// TIA Portal V20 program export: 31 tag tables, 33 data types, 19 data blocks, 74 code blocks (in call order from the OBs), 22 instance data blocks

VAR_GLOBAL   // PLC tag table "Default tag table"
   System_Byte AT %MB1 : Byte;
   FirstScan AT %M1.0 : Bool;
   DiagStatusUpdate AT %M1.1 : Bool;
   AlwaysTRUE AT %M1.2 : Bool;
   AlwaysFALSE AT %M1.3 : Bool;
   Clock_Byte AT %MB0 : Byte;
   Clock_10Hz AT %M0.0 : Bool;
   Clock_5Hz AT %M0.1 : Bool;
   "Clock_2.5Hz" AT %M0.2 : Bool;
   Clock_2Hz AT %M0.3 : Bool;
   "Clock_1.25Hz" AT %M0.4 : Bool;
   Clock_1Hz AT %M0.5 : Bool;
   "Clock_0.625Hz" AT %M0.6 : Bool;
   "Clock_0.5Hz" AT %M0.7 : Bool;
   startBit AT %M100.0 : Bool;
   stopBit AT %M100.1 : Bool;
   ResetBit AT %M100.2 : Bool;
END_VAR

VAR_GLOBAL   // PLC tag table "Tag table_1"
END_VAR

VAR_GLOBAL   // PLC tag table "Default tag table_1"
END_VAR

VAR_GLOBAL   // PLC tag table "ConvConstantEmptyLine"
END_VAR
VAR_GLOBAL CONSTANT   // user constants
   minEmptyLine : Int := 2001;
   maxEmptyLine : Int := 2109;
   "J1.1.1" : Int := 2001;   // J1.1.1
   "J1.1.2" : Int := 2002;   // J1.1.2
   "J1.1.3" : Int := 2003;   // J1.1.3
   "J1.1.4" : Int := 2004;   // J1.1.4
   "J1.1.5" : Int := 2005;   // J1.1.5
   "J1.1.6" : Int := 2006;   // J1.1.6
   "J1.1.7" : Int := 2007;   // J1.1.7
   "J1.1.8" : Int := 2008;   // J1.1.8
   "J1.1.9" : Int := 2009;   // J1.1.9
   "J1.1.10" : Int := 2010;   // J1.1.10
   "J1.1.11" : Int := 2011;   // J1.1.11
   "J1.1.12" : Int := 2012;   // J1.1.12
   "J1.1.13" : Int := 2013;   // J1.1.13
   "J1.1.14" : Int := 2014;   // J1.1.14
   "J1.1.15" : Int := 2015;   // J1.1.15
   "J1.2.1" : Int := 2016;   // J1.2.1
   "J1.2.2" : Int := 2017;   // J1.2.2
   "J1.2.3" : Int := 2018;   // J1.2.3 Staright for Merger1
   "J2.1.1" : Int := 2019;   // J2.1.1
   "J2.1.2" : Int := 2020;   // J2.1.2
   "J2.1.3" : Int := 2021;   // J2.1.3
   "J2.1.4" : Int := 2022;   // J2.1.4
   "J2.1.5" : Int := 2023;   // J2.1.5
   "J2.1.6" : Int := 2024;   // J2.1.6
   "J2.1.7" : Int := 2025;   // J2.1.7
   "J2.1.8" : Int := 2026;   // J2.1.8
   "J2.1.9" : Int := 2027;   // J2.1.9
   "J2.1.10" : Int := 2028;   // J2.1.10
   "J2.1.11" : Int := 2029;   // J2.1.11
   "J2.1.12" : Int := 2030;   // J2.1.12
   "J2.1.13" : Int := 2031;   // J2.1.13
   "J2.1.14" : Int := 2032;   // J2.1.14
   "J2.1.15" : Int := 2033;   // J2.1.15
   "J2.2.1" : Int := 2034;   // J2.2.1
   "J2.2.2" : Int := 2035;   // J2.2.2
   "J2.3.1" : Int := 2036;   // J2.3.1
   "J2.4.1" : Int := 2037;   // J2.4.1 Arm for Merger1
   "J1.2.4" : Int := 2038;   // J1.2.4 Merger 1
   "J1.2.5" : Int := 2039;   // J1.2.5
   "J1.3.1" : Int := 2040;   // J1.3.1
   "J1.3.2" : Int := 2041;   // J1.3.2
   "J1.4.1" : Int := 2042;   // J1.4.1
   "J1.4.2" : Int := 2043;   // J1.4.2
   "J1.4.3" : Int := 2044;   // J1.4.3
   "J1.4.4" : Int := 2045;   // J1.4.4
   "J1.4.5" : Int := 2046;   // J1.4.5
   "J1.4.6" : Int := 2047;   // J1.4.6
   "J1.4.7" : Int := 2048;   // J1.4.7
   "J1.5.1" : Int := 2049;   // J1.5.1
   "J1.5.2" : Int := 2050;   // J1.5.2
   "J1.5.3" : Int := 2051;   // J1.5.3
   "J1.5.4" : Int := 2052;   // J1.5.4
   "J1.7.1" : Int := 2053;   // J1.7.1 (Go straight )
   "J1.7.2" : Int := 2054;   // J1.7.2
   "J1.8.1" : Int := 2055;   // J1.8.1
   "J1.8.2" : Int := 2056;   // J1.8.2
   "J1.9.1" : Int := 2057;   // J1.9.1
   "J1.10.1" : Int := 2058;   // J1.10.1
   "J1.11.1" : Int := 2059;   // J1.11.1
   "J1.11.2" : Int := 2060;   // J1.11.2
   "J1.11.3" : Int := 2061;   // J1.11.3
   "J1.11.4" : Int := 2062;   // J1.11.4
   "J1.11.5" : Int := 2063;   // J1.11.5
   "J1.11.6" : Int := 2064;   // J1.11.6
   "J1.11.7" : Int := 2065;   // J1.11.7
   "J1.11.8" : Int := 2066;   // J1.11.8
   "J1.11.9" : Int := 2067;   // J1.11.9
   "J1.11.10" : Int := 2068;   // J1.11.10
   "J1.11.11" : Int := 2069;   // J1.11.11
   "J1.11.12" : Int := 2070;   // J1.11.12
   "J1.11.13" : Int := 2071;   // J1.11.13
   "K1.1.1" : Int := 2072;   // K1.1.1 (Go Left)
   "K1.2.1" : Int := 2073;   // K1.2.1
   "K1.3.1" : Int := 2074;   // K1.3.1
   "K1.4.1" : Int := 2075;   // K1.4.1
   "K1.4.2" : Int := 2076;   // K1.4.2
   "K1.4.3" : Int := 2077;   // K1.4.3
   "K1.4.4" : Int := 2078;   // K1.4.4
   "K1.4.5" : Int := 2079;   // K1.4.5
   "K1.4.6" : Int := 2080;   // K1.4.6
   "K1.4.7" : Int := 2081;   // K1.4.7
   "K1.4.8" : Int := 2082;   // K1.4.8
   "K1.4.9" : Int := 2083;   // K1.4.9
   "K1.4.10" : Int := 2084;   // K1.4.10
   "K1.5.1" : Int := 2085;   // K1.5.1
   "K1.5.2" : Int := 2086;   // K1.5.2
   "K1.5.3" : Int := 2087;   // K1.5.3
   "K1.5.4" : Int := 2088;   // K1.5.4
   "K1.5.5" : Int := 2089;   // K1.5.5
   "K1.5.6" : Int := 2090;   // K1.5.6
   "K1.5.7" : Int := 2091;   // K1.5.7
   "K1.5.8" : Int := 2092;   // K1.5.8
   "K1.6.1" : Int := 2093;   // K1.6.1
   "K1.6.2" : Int := 2094;   // K1.6.2
   "K1.7.1" : Int := 2095;   // K1.7.1
   "K1.7.2" : Int := 2096;   // K1.7.2
   "K1.8.1" : Int := 2097;   // K1.8.1
   "K1.8.2" : Int := 2098;   // K1.8.2
   "K1.8.3" : Int := 2099;   // K1.8.3
   "K1.9.1" : Int := 2100;   // K1.9.1
   "K1.9.2" : Int := 2101;   // K1.9.2
   "K1.9.3" : Int := 2102;   // K1.9.3
   "K1.9.4" : Int := 2103;   // K1.9.4
   "K1.9.5" : Int := 2104;   // K1.9.5
   "K1.9.6" : Int := 2105;   // K1.9.6
   "K1.9.7" : Int := 2106;   // K1.9.7
   "K1.10.1" : Int := 2107;   // K1.10.1
   "J1.6.1" : Int := 2108;   // Mabs J1.6.1
   "J1.6.2" : Int := 2109;   // Mabs J1.6.2
END_VAR

VAR_GLOBAL   // PLC tag table "MabsEmptyLine"
   "MABS_J1.6.1_IN" AT %I839.0 : "Global.IB_P01_02_03_in_64bytes_struct";
   "MABS_J1.6.1_Out" AT %Q761.0 : "Global.IB_P01_02_03_out_64bytes_struct";
   "MABS_J1.6.2_IN" AT %I903.0 : "Global.IB_P01_02_03_in_64bytes_struct";
   "MABS_J1.6.2_Out" AT %Q825.0 : "Global.IB_P01_02_03_out_64bytes_struct";
END_VAR

VAR_GLOBAL   // PLC tag table "ASi Alarm"
   "BW_ASi23 -MCC100 -210KE3 -ConfigErr_Circuit1_Slave(16-31)A" AT %IW2366 : Word;
   "BW_ASi23 -MCC100 -210KE3 -ConfigErr_Circuit1_Slave(16-31)B" AT %IW2370 : Word;
   "BW_ASi23 -MCC100 -210KE3 -PeriErr_Circuit1_Slave(16-31)A" AT %IW2374 : Word;
   "BW_ASi23 -MCC100 -210KE3 -PeriErr_Circuit1_Slave(16-31)B" AT %IW2378 : Word;
   "BW_ASi23 -MCC100 -210KE3 -ConfigErr_Circuit2_Slave(0-15)A" AT %IW2380 : Word;
   "BW_ASi23 -MCC100 -210KE3 -ConfigErr_Circuit2_Slave(16-31)A" AT %IW2382 : Word;
   "BW_ASi23 -MCC100 -210KE3 -ConfigErr_Circuit2_Slave(0-15)B" AT %IW2384 : Word;
   "BW_ASi23 -MCC100 -210KE3 -ConfigErr_Circuit2_Slave(16-31)B" AT %IW2386 : Word;
   "BW_ASi23 -MCC100 -210KE3 -PeriErr_Circuit2_Slave(0-15)A" AT %IW2388 : Word;
   "BW_ASi23 -MCC100 -210KE3 -PeriErr_Circuit2_Slave(16-31)A" AT %IW2390 : Word;
   "BW_ASi23 -MCC100 -210KE3 -PeriErr_Circuit2_Slave(0-15)B" AT %IW2392 : Word;
   "BW_ASi23 -MCC100 -210KE3 -PeriErr_Circuit2_Slave(16-31)B" AT %IW2394 : Word;
   "BW_ASi23 -MCC100 -210KE3 -ConfigErr_Circuit1_Slave(0-15)A" AT %IW2364 : Word;
   "BW_ASi23 -MCC100 -210KE3 -ConfigErr_Circuit1_Slave(0-15)B" AT %IW2368 : Word;
   "BW_ASi23 -MCC100 -210KE3 -PeriErr_Circuit1_Slave(0-15)A" AT %IW2372 : Word;
   "BW_ASi23 -MCC100 -210KE3 -PeriErr_Circuit1_Slave(0-15)B" AT %IW2376 : Word;
END_VAR

VAR_GLOBAL   // PLC tag table "ASi"
   "ASiGW-MCC100-bw23-C1: Input" AT %I2300.0 : "tASiGW-MCC100-bw23-C1: Input";
   "ASiGW-MCC100-bw23-C1: Output" AT %Q2300.0 : "tASiGW-MCC100-bw23-C1: Output";
   "ASiGW-MCC100-bw23-C1: ConfigErr" AT %I2364.0 : "Config/PeriErr";
   "ASiGW-MCC100-bw23-C1: PeriErr" AT %I2372.0 : "Config/PeriErr";
END_VAR

VAR_GLOBAL   // PLC tag table "Circuit Breaker"
END_VAR

VAR_GLOBAL   // PLC tag table "ConvConstant"
END_VAR
VAR_GLOBAL CONSTANT   // user constants
   gMinA1 : Int := 1001;
   gMaxA1 : Int := 1002;
   gMinB1 : Int := 2001;
   gMaxB1 : Int := 2002;
   gMinC1 : Int := 3001;
   gMaxC1 : Int := 3054;
   gMinD1 : Int := 4001;
   gMaxD1 : Int := 4002;
END_VAR

VAR_GLOBAL   // PLC tag table "DM262"
   "Dataman-TriggerEnable" AT %Q10.0 : Bool;
   "Dataman-Trigger" AT %Q10.1 : Bool;
   "Dataman-TriggerReady" AT %I10.0 : Bool;
   "Dataman-TriggerAck" AT %I10.1 : Bool;
   "Dataman-Acquiring" AT %I10.2 : Bool;
   "Dataman-MissedAcq" AT %I10.3 : Bool;
   "Dataman-TriggerID" AT %IW11 : Word;
   "Dataman-BufferResultsEnable" AT %Q11.0 : Bool;
   "Dataman-ResultsAck" AT %Q11.1 : Bool;
   "Dataman-Decoding" AT %I13.0 : Bool;
   "Dataman-Decode Complete" AT %I13.1 : Bool;
   "Dataman-Results Buffer Overrun" AT %I13.2 : Bool;
   "Dataman-Results Available" AT %I13.3 : Bool;
   "Dataman-General Fault" AT %I13.7 : Bool;
   "Dataman-Train Code" AT %Q12.0 : Bool;
   "Dataman-Train Match String" AT %Q12.1 : Bool;
   "Dataman-Train Focus" AT %Q12.2 : Bool;
   "Dataman-Train Brightness" AT %Q12.3 : Bool;
   "Dataman-Untrain" AT %Q12.4 : Bool;
   "Dataman-Execute DMCC" AT %Q12.6 : Bool;
   "Dataman-Set Match String" AT %Q12.7 : Bool;
   "Dataman-Train Code Ack" AT %I14.0 : Bool;
   "Dataman-Train Match String Ack" AT %I14.1 : Bool;
   "Dataman-Train Focus Ack" AT %I14.2 : Bool;
   "Dataman-Train Brightness Ack" AT %I14.3 : Bool;
   "Dataman-Untrain Ack" AT %I14.4 : Bool;
   "Dataman-Execute DMCC Ack" AT %I14.6 : Bool;
   "Dataman-Set Match String Ack" AT %I14.7 : Bool;
   "Dataman-UserData Option" AT %QW13 : Word;
   "Dataman-UserData Length" AT %QW15 : Word;
   "Dataman-UserData[0]" AT %QB17 : Byte;
   "Dataman-UserData[1]" AT %QB18 : Byte;
   "Dataman-UserData[2]" AT %QB19 : Byte;
   "Dataman-UserData[3]" AT %QB20 : Byte;
   "Dataman-UserData[4]" AT %QB21 : Byte;
   "Dataman-UserData[5]" AT %QB22 : Byte;
   "Dataman-UserData[6]" AT %QB23 : Byte;
   "Dataman-UserData[7]" AT %QB24 : Byte;
   "Dataman-UserData[8]" AT %QB25 : Byte;
   "Dataman-UserData[9]" AT %QB26 : Byte;
   "Dataman-UserData[10]" AT %QB27 : Byte;
   "Dataman-UserData[11]" AT %QB28 : Byte;
   "Dataman-UserData[12]" AT %QB29 : Byte;
   "Dataman-UserData[13]" AT %QB30 : Byte;
   "Dataman-UserData[14]" AT %QB31 : Byte;
   "Dataman-UserData[15]" AT %QB32 : Byte;
   "Dataman-ResultID" AT %IW15 : Word;
   "Dataman-Result Code" AT %IW18 : Word;
   "Dataman-Read / No Read" AT %I18.0 : Bool;
   "Dataman-Validated / Not Validated" AT %I18.1 : Bool;
   "Dataman-Verified / Not Verified" AT %I18.2 : Bool;
   "Dataman-Acquisition Trigger Overrun" AT %I18.3 : Bool;
   "Dataman-Acquisition Buffer Overflow" AT %I18.4 : Bool;
   "Dataman-Result Extended" AT %IW19 : Word;
   "Dataman-Result Length" AT %IW21 : Word;
   "Dataman-InspectionResults[0]" AT %IB23 : Byte;
   "Dataman-InspectionResults[1]" AT %IB24 : Byte;
   "Dataman-InspectionResults[2]" AT %IB25 : Byte;
   "Dataman-InspectionResults[3]" AT %IB26 : Byte;
   "Dataman-InspectionResults[4]" AT %IB27 : Byte;
   "Dataman-InspectionResults[5]" AT %IB28 : Byte;
   "Dataman-InspectionResults[6]" AT %IB29 : Byte;
   "Dataman-InspectionResults[7]" AT %IB30 : Byte;
   "Dataman-InspectionResults[8]" AT %IB31 : Byte;
   "Dataman-InspectionResults[9]" AT %IB32 : Byte;
   "Dataman-InspectionResults[10]" AT %IB33 : Byte;
   "Dataman-InspectionResults[11]" AT %IB34 : Byte;
   "Dataman-InspectionResults[12]" AT %IB35 : Byte;
   "Dataman-InspectionResults[13]" AT %IB36 : Byte;
   "Dataman-InspectionResults[14]" AT %IB37 : Byte;
   "Dataman-InspectionResults[15]" AT %IB38 : Byte;
   "Result Data" AT %I23.0 : "Global.BarCode";
   "User Data" AT %Q17.0 : "Global.BarCode";
END_VAR

VAR_GLOBAL   // PLC tag table "Default tag table_3"
END_VAR

VAR_GLOBAL   // PLC tag table "Klaxon"
END_VAR

VAR_GLOBAL   // PLC tag table "SSR"
END_VAR

VAR_GLOBAL   // PLC tag table "Safety"
END_VAR

VAR_GLOBAL   // PLC tag table "ConvConstantA1"
END_VAR
VAR_GLOBAL CONSTANT   // user constants
   minA1 : Int := 1001;
   maxA1 : Int := 1002;
END_VAR

VAR_GLOBAL   // PLC tag table "ConvConstantB1"
END_VAR
VAR_GLOBAL CONSTANT   // user constants
   minB1 : Int := 2001;
   maxB1 : Int := 2002;
END_VAR

VAR_GLOBAL   // PLC tag table "Default tag table_2"
END_VAR

VAR_GLOBAL   // PLC tag table "ConvConstantC1"
END_VAR
VAR_GLOBAL CONSTANT   // user constants
   minC1 : Int := 3001;
   maxC1 : Int := 3054;
   "Conveyor_C1.1.1" : Int := 3001;
   "Conveyor_C1.1.2" : Int := 3002;
   "Conveyor_C1.1.3" : Int := 3003;
   "MABS_C1.2.1" : Int := 3051;
   "MABS_C1.2.2" : Int := 3052;
   "Conveyor_C1.9.1" : Int := 3031;
   "Conveyor_C1.10.1" : Int := 3032;
   "Conveyor_C1.11.1" : Int := 3033;
   "Conveyor_C1.11.2" : Int := 3034;
   "Conveyor_C1.12.1" : Int := 3035;
   "Conveyor_C1.12.2" : Int := 3036;
   "Conveyor_C1.12.3" : Int := 3037;
   "Transfer_C1.13.1" : Int := 3053;
   "Transfer_C1.14.1" : Int := 3054;
   "Conveyor_C1.15.2" : Int := 3038;
   "Conveyor_C1.15.3" : Int := 3039;
   "Conveyor_C1.15.4" : Int := 3040;
   "Conveyor_C1.16.1" : Int := 3041;
   "Conveyor_C1.18.1" : Int := 3042;
   "Conveyor_C1.18.2" : Int := 3043;
   "Conveyor_C1.18.3" : Int := 3044;
   "Conveyor_C1.18.4" : Int := 3045;
   "Conveyor_C1.18.5" : Int := 3046;
   "Conveyor_C1.18.6" : Int := 3047;
   "Conveyor_C1.18.7" : Int := 3048;
   "Conveyor_C1.19.1" : Int := 3049;
   "Conveyor_C1.20.2" : Int := 3050;
   "Conveyor_C1.3.1" : Int := 3004;
   "Conveyor_C1.3.2" : Int := 3005;
   "Conveyor_C1.3.3" : Int := 3006;
   "Conveyor_C1.3.4" : Int := 3007;
   "Conveyor_C1.3.5" : Int := 3008;
   "Conveyor_C1.3.6" : Int := 3009;
   "Conveyor_C1.3.7" : Int := 3010;
   "Conveyor_C1.3.8" : Int := 3011;
   "Conveyor_C1.3.9" : Int := 3012;
   "Conveyor_C1.3.10" : Int := 3013;
   "Conveyor_C1.4.1" : Int := 3014;
   "Conveyor_C1.4.2" : Int := 3015;
   "Conveyor_C1.4.3" : Int := 3016;
   "Conveyor_C1.4.4" : Int := 3017;
   "Conveyor_C1.5.1" : Int := 3018;
   "Conveyor_C1.6.1" : Int := 3019;
   "Conveyor_C1.6.2" : Int := 3020;
   "Conveyor_C1.7.1" : Int := 3021;
   "Conveyor_C1.7.2" : Int := 3022;
   "Conveyor_C1.7.3" : Int := 3023;
   "Conveyor_C1.7.4" : Int := 3024;
   "Conveyor_C1.7.5" : Int := 3025;
   "Conveyor_C1.7.6" : Int := 3026;
   "Conveyor_C1.7.7" : Int := 3027;
   "Conveyor_C1.7.8" : Int := 3028;
   "Conveyor_C1.7.9" : Int := 3029;
   "Conveyor_C1.7.10" : Int := 3030;
END_VAR

VAR_GLOBAL   // PLC tag table "Default tag table_4"
   sensor AT %I0.0 : Bool;
END_VAR

VAR_GLOBAL   // PLC tag table "MABS"
   "MABS_C1.2.1_IN" AT %I100.0 : "IB_P01/02/03_in_64bytes_struct";
   "MABS_C1.2.1_Out" AT %I200.0 : "IB_P01/02/03_out_64bytes_struct";
   "MABS_C1.2.2_IN" AT %I300.0 : "IB_P01/02/03_in_64bytes_struct";
   "MABS_C1.2.2_Out" AT %I400.0 : "IB_P01/02/03_out_64bytes_struct";
END_VAR

VAR_GLOBAL   // PLC tag table "ConvConstantD1"
END_VAR
VAR_GLOBAL CONSTANT   // user constants
   minD1 : Int := 4001;
   maxD1 : Int := 4002;
END_VAR

VAR_GLOBAL   // PLC tag table "Default tag table_6"
END_VAR

VAR_GLOBAL   // PLC tag table "ConvConstantPackedLine"
END_VAR
VAR_GLOBAL CONSTANT   // user constants
   minPackedLine : Int := 3001;
   maxPackedLine : Int := 3040;
   "G1.1.1" : Int := 3001;   // G1.1.1
   "G1.1.2" : Int := 3002;   // G1.1.2
   "G1.1.3" : Int := 3003;   // G1.1.3
   "G1.1.4" : Int := 3004;   // G1.1.4
   "G1.1.5" : Int := 3005;   // G1.1.5
   "G1.1.6" : Int := 3006;   // G1.1.6
   "G1.1.7" : Int := 3007;   // G1.1.7
   "G1.1.8" : Int := 3008;   // G1.1.8
   "G1.1.9" : Int := 3009;   // G1.1.9
   "G1.1.10" : Int := 3010;   // G1.1.10
   "G1.1.11" : Int := 3011;   // G1.1.11
   "G1.1.12" : Int := 3012;   // G1.1.12
   "G1.1.13" : Int := 3013;   // G1.1.13
   "G1.1.14" : Int := 3014;   // G1.1.14
   "G1.1.15" : Int := 3015;   // G1.1.15
   "G1.1.16" : Int := 3016;   // G1.1.16
   "G1.1.17" : Int := 3017;   // G1.1.17
   "G1.1.18" : Int := 3018;   // G1.1.18
   "G1.1.19" : Int := 3019;   // G1.1.19
   "G1.2.1" : Int := 3020;   // G1.2.1
   "G1.2.2" : Int := 3021;   // G1.2.2
   "G1.3.1" : Int := 3022;   // G1.3.1
   "G1.4.1" : Int := 3023;   // G1.4.1
   "G1.4.2" : Int := 3024;   // G1.4.2
   "G1.4.3" : Int := 3025;   // G1.4.3
   "G1.4.4" : Int := 3026;   // G1.4.4
   "G1.4.5" : Int := 3027;   // G1.4.5
   "G1.4.6" : Int := 3028;   // G1.4.6
   "G1.5.1" : Int := 3029;   // G1.5.1
   "G1.5.2" : Int := 3030;   // G1.5.2
   "G1.5.3" : Int := 3031;   // G1.5.3
   "G1.5.4" : Int := 3032;   // G1.5.4
   "G1.5.5" : Int := 3033;   // G1.5.5
   "G1.5.6" : Int := 3034;   // G1.5.6
   "G1.6.1" : Int := 3035;   // G1.6.1
   "G1.6.2" : Int := 3036;   // G1.6.2
   "G1.7.1" : Int := 3037;   // G1.7.1
   "G1.7.2" : Int := 3038;   // G1.7.2
   "G1.7.3" : Int := 3039;   // G1.7.3
   "G1.7.4" : Int := 3040;   // G1.7.4
END_VAR

VAR_GLOBAL   // PLC tag table "ConvConstantProductionLine"
END_VAR
VAR_GLOBAL CONSTANT   // user constants
   minProductionLine : Int := 1001;
   maxProductionLine : Int := 1192;
   "A1.1.1" : Int := 1001;
   "A1.1.2" : Int := 1002;
   "A1.1.3" : Int := 1003;
   "A1.1.4" : Int := 1004;
   "A1.1.5" : Int := 1005;
   "A1.1.6" : Int := 1006;
   "A1.1.7" : Int := 1007;
   "A1.1.8" : Int := 1008;
   "A1.1.9" : Int := 1009;
   "A1.1.10" : Int := 1010;
   "A1.1.11" : Int := 1011;
   "A1.1.12" : Int := 1012;
   "A1.1.13" : Int := 1013;
   "A1.1.14" : Int := 1014;
   "A1.2.1" : Int := 1015;   // //A1.2.1 (DP1)
   "A1.3.1" : Int := 1016;
   "A1.4.1" : Int := 1017;
   "A1.5.1" : Int := 1018;
   "A1.5.2" : Int := 1019;
   "A1.5.3" : Int := 1020;
   "A1.7.1" : Int := 1021;   // // A1.7.1 (Go Straight DP1)
   "A1.7.2" : Int := 1022;   // //A1.7.2 Straight for Merger1
   "A1.7.3" : Int := 1023;
   "A1.7.4" : Int := 1024;   // //A1.7.4 (DP4)
   "A1.7.5" : Int := 1025;
   "A1.7.6" : Int := 1026;
   "A1.8.1" : Int := 1027;
   "A1.10.1" : Int := 1028;   // // A1.9.1 (Go Straight DP4)
   "A1.10.2" : Int := 1029;   // //A1.9.2 Straight for Merger2
   "A1.10.3" : Int := 1030;   // // A1.9.3 Merger2
   "A1.10.4" : Int := 1031;
   "A1.10.5" : Int := 1032;
   "A1.10.6" : Int := 1033;
   "A1.10.7" : Int := 1034;
   "A1.10.8" : Int := 1035;
   "A1.10.9" : Int := 1036;
   "A1.10.10" : Int := 1037;
   "A1.10.11" : Int := 1038;
   "A1.10.12" : Int := 1039;
   "A1.10.13" : Int := 1040;
   "A1.11.1" : Int := 1041;
   "A1.11.2" : Int := 1042;
   "A1.12.1" : Int := 1043;
   "A1.12.2" : Int := 1044;
   "A1.14.1" : Int := 1045;   // // A1.13.1 (Go straight TR_A1.12.1)
   "A1.14.2" : Int := 1046;
   "A1.14.3" : Int := 1047;
   "A1.14.4" : Int := 1048;
   "A1.14.5" : Int := 1049;
   "A1.14.6" : Int := 1050;
   "A1.14.7" : Int := 1051;
   "A1.14.8" : Int := 1052;
   "A1.14.9" : Int := 1053;
   "A1.14.10" : Int := 1054;
   "A1.14.11" : Int := 1055;
   "A1.14.12" : Int := 1056;
   "A1.14.13" : Int := 1057;
   "A1.14.14" : Int := 1058;
   "A1.14.15" : Int := 1059;
   "A2.2.1" : Int := 1071;   // // A1.17.2 (Go straight TR_A2.1.1)
   "A2.2.2" : Int := 1072;
   "A2.2.3" : Int := 1073;
   "A2.2.4" : Int := 1074;
   "A2.2.5" : Int := 1075;
   "A2.2.6" : Int := 1076;
   "A2.2.7" : Int := 1077;
   "A2.2.8" : Int := 1078;
   "A2.2.9" : Int := 1079;
   "A2.2.10" : Int := 1080;
   "A2.2.11" : Int := 1081;
   "A2.2.12" : Int := 1082;
   "A2.2.13" : Int := 1083;
   "A2.2.14" : Int := 1084;
   "A2.2.15" : Int := 1085;
   "B1.1.1" : Int := 1097;   // // B1.1.1 (Go Right DP1)
   "B1.2.1" : Int := 1098;
   "B1.3.1" : Int := 1099;
   "B1.3.2" : Int := 1100;
   "B1.3.3" : Int := 1101;
   "B1.4.1" : Int := 1102;
   "B1.4.2" : Int := 1103;
   "B1.5.1" : Int := 1104;
   "B1.7.1" : Int := 1105;   // // B1.7.1 (Go straight TR_A1.7.1)
   "B1.7.2" : Int := 1106;
   "B1.7.3" : Int := 1107;
   "B1.8.1" : Int := 1108;
   "B1.8.2" : Int := 1109;
   "B1.8.3" : Int := 1110;
   "B1.9.1" : Int := 1111;   // // B1.9.1 (DP2)
   "B1.9.2" : Int := 1112;
   "B1.11.1" : Int := 1113;   // // B1.11.1 (Go straight TR_B1.11.1)
   "B1.11.2" : Int := 1114;
   "B1.11.3" : Int := 1115;
   "B1.11.4" : Int := 1116;
   "B1.12.1" : Int := 1117;
   "B1.12.2" : Int := 1118;
   "B1.15.1" : Int := 1119;   // // B1.18.1 (Go straight TR_B1.17.1)
   "B1.15.2" : Int := 1120;
   "B1.16.1" : Int := 1121;
   "B1.16.2" : Int := 1122;
   "B1.16.3" : Int := 1123;
   "B1.16.4" : Int := 1124;
   "B1.16.5" : Int := 1125;
   "B1.16.6" : Int := 1126;
   "B1.16.7" : Int := 1127;
   "B1.16.8" : Int := 1128;
   "B1.17.1" : Int := 1129;   // // B1.20.1 (DP3)
   "B1.17.2" : Int := 1130;
   "B1.17.3" : Int := 1131;
   "B1.17.4" : Int := 1132;
   "B1.19.1" : Int := 1133;
   "B1.20.1" : Int := 1134;
   "B1.20.2" : Int := 1135;
   "B1.21.1" : Int := 1136;
   "B1.21.2" : Int := 1137;
   "B1.21.3" : Int := 1138;
   "B1.22.1" : Int := 1139;
   "B1.23.1" : Int := 1140;   // //B1.28.1 Arm for Merger1
   "C1.2.2" : Int := 1141;   // // C1.1.2 (Go Right TR_C1.1.3)
   "C1.2.1" : Int := 1142;
   "C1.4.1" : Int := 1143;   // // C1.1.4 (Go Left TR_C1.1.3)
   "C1.4.2" : Int := 1144;
   "D1.1.1" : Int := 1145;   // // D1.1.1 (Go Right DP4)
   "D1.2.1" : Int := 1146;
   "D1.3.1" : Int := 1147;
   "D1.4.1" : Int := 1148;
   "D1.5.1" : Int := 1149;
   "D1.6.1" : Int := 1150;
   "D1.7.1" : Int := 1151;
   "D1.7.2" : Int := 1152;
   "D1.7.3" : Int := 1153;
   "D1.7.4" : Int := 1154;
   "D1.7.5" : Int := 1155;
   "D1.7.6" : Int := 1156;
   "D1.7.7" : Int := 1157;
   "D1.7.8" : Int := 1158;
   "D1.7.9" : Int := 1159;
   "D1.7.10" : Int := 1160;
   "D1.8.1" : Int := 1161;
   "D1.8.2" : Int := 1162;
   "D1.8.3" : Int := 1163;
   "D1.11.1" : Int := 1164;
   "D1.11.2" : Int := 1165;
   "D1.11.3" : Int := 1166;
   "D1.12.1" : Int := 1167;
   "D1.12.2" : Int := 1168;
   "D1.12.3" : Int := 1169;   // //End
   "E1.1.2" : Int := 1171;
   "E1.1.3" : Int := 1172;
   "E1.1.4" : Int := 1173;
   "E1.2.1" : Int := 1174;
   "E1.3.1" : Int := 1175;
   "E1.4.1" : Int := 1176;
   "E1.5.1" : Int := 1177;
   "E1.6.1" : Int := 1178;   // //E1.6.1 Arm for Merger2
   "A1.9.1" : Int := 1179;   // // Mabs A1.8.1
   "A1.9.2" : Int := 1180;   // // Mabs A1.8.2
   "A1.6.1" : Int := 1181;   // // Mabs A1.6.1
   "A1.6.2" : Int := 1182;   // // Mabs A1.6.2
   "A1.13.1" : Int := 1183;   // // Transfer A1.12.1
   "A2.1.1" : Int := 1184;   // // Transfer A2.1.1
   "B1.6.1" : Int := 1185;   // // Transfer B1.6.1
   "B1.10.1" : Int := 1186;   // // Transfer B1.10.1
   "B1.13.1" : Int := 1187;   // // Transfer B1.16.1
   "B1.14.1" : Int := 1188;   // // Transfer B1.17.1
   "B1.18.1" : Int := 1189;   // // Transfer B1.21.1
   "C1.3.1" : Int := 1190;   // //Transfer C1.1.3
   "D1.9.1" : Int := 1191;   // //Transfer D1.8.1
   "D1.10.1" : Int := 1192;   // //Transfer D1.9.1
   "A1.14.16" : Int := 1060;
   "A1.14.17" : Int := 1061;
   "A1.14.18" : Int := 1062;
   "A1.14.19" : Int := 1063;
   "A1.14.20" : Int := 1064;
   "A1.14.21" : Int := 1065;
   "A1.14.22" : Int := 1066;
   "A1.14.23" : Int := 1067;
   "A1.14.24" : Int := 1068;
   "A2.2.16" : Int := 1086;
   "A2.2.17" : Int := 1087;
   "A2.2.18" : Int := 1088;
   "A2.2.19" : Int := 1089;
   "A2.2.20" : Int := 1090;
   "A2.2.21" : Int := 1091;
   "A2.2.22" : Int := 1092;
   "A2.2.23" : Int := 1093;
   "A2.2.24" : Int := 1094;
   "E1.1.1" : Int := 1170;
   "A1.14.25" : Int := 1069;
   "A1.14.26" : Int := 1070;
   "A2.2.25" : Int := 1095;
   "A2.2.26" : Int := 1096;
END_VAR

VAR_GLOBAL   // PLC tag table "Default tag table_5"
END_VAR

VAR_GLOBAL   // PLC tag table "IMC84"
   "IMC84Sensor -1" AT %I583.0 : Bool;   // High = Sensor active (input type and polarity can be configured)
   IMC84Sensor_2 AT %I583.1 : Bool;   // High = Sensor active (input type and polarity can be configured)
   IMC84Sensor_3 AT %I583.2 : Bool;   // High = Sensor active (input type and polarity can be configured)
   IMC84Sensor_4 AT %I583.3 : Bool;   // High = Sensor active (input type and polarity can be configured)
   IMC84Sensor_5 AT %I583.4 : Bool;
   IMC84Sensor_6 AT %I583.5 : Bool;
   IMC84Sensor_7 AT %I583.6 : Bool;
   IMC84Sensor_8 AT %I583.7 : Bool;
   IMC84IO1 AT %I584.0 : Bool;   // Digital I/O PLC Input PLC Output
   IMC84IO2 AT %I584.1 : Bool;   // Digital I/O PLC Input PLC Output
   IMC84IO3 AT %I584.2 : Bool;   // Digital I/O PLC Input PLC Output
   IMC84IO4 AT %I584.3 : Bool;   // Digital I/O PLC Input PLC Output
   IMC84IO5 AT %I584.4 : Bool;
   IMC84IO6 AT %I584.5 : Bool;
   IMC84IO7 AT %I584.6 : Bool;
   IMC84IO8 AT %I584.7 : Bool;
   "IMC84MotorStateErrorRD -G1.4.3" AT %I585.0 : Bool;   // High = Motor Error; Low = Motor OK
   "IMC84MotorStateErrorRD -G1.4.2" AT %I585.1 : Bool;   // High = Motor Error; Low = Motor OK
   "IMC84MotorStateErrorRD -G1.4.1" AT %I585.2 : Bool;   // High = Motor Error; Low = Motor OK
   "IMC84MotorStateErrorRD_G1.3.1" AT %I585.3 : Bool;   // High = Motor Error; Low = Motor OK
   "IMC84MotorStateSpeedRD -G1.4.3" AT %IB586 : SInt;   // Speed 0–100 ( 0 = Stop, 100 = max speed), negative sign reverses the turning direction
   "IMC84MotorStateSpeedRD -G1.4.2" AT %IB587 : SInt;   // Speed 0–100 ( 0 = Stop, 100 = max speed), negative sign reverses the turning direction
   "IMC84MotorStateSpeedRD -G1.4.1" AT %IB588 : SInt;   // Speed 0–100 ( 0 = Stop, 100 = max speed), negative sign reverses the turning direction
   "IMC84MotorStateSpeedRD_G1.3.1" AT %IB589 : SInt;   // Speed 0–100 ( 0 = Stop, 100 = max speed), negative sign reverses the turning direction
   "IMC84MotorCurrentRD -G1.4.3" AT %IW591 : Int;   // Average current in mA
   "IMC84MotorCurrentRD -G1.4.2" AT %IW593 : Int;   // Average current in mA
   "IMC84MotorCurrentRD -G1.4.1" AT %IW595 : Int;   // Average current in mA
   "IMC84MotorCurrentRD_G1.3.1" AT %IW597 : Int;   // Average current in mA
   "IMC84Voltage(MotorPower)" AT %IW599 : Int;   // Voltage „Motor Power“ in mV
   "IMC84Voltage(Sensors)" AT %IW601 : Int;   // Voltage „Power Logic + Sensors“ in mV
   IMC84Temperature AT %IW603 : Int;   // Temperature in 0,1 C
   IMC84SystemUpTime AT %ID605 : DInt;   // Operating time in seconds since the last start/restart
   "IMC84DigitalOutputRD -G1.4.3" AT %Q64.0 : Bool;
   "IMC84DigitalOutputRD -G1.4.2" AT %Q64.1 : Bool;
   "IMC84DigitalOutputRD -G1.4.1" AT %Q64.2 : Bool;
   "IMC84DigitalOutputRD_G1.3.1" AT %Q64.3 : Bool;
   "IMC84MotorTargetSpeedRD -G1.4.3" AT %QB65 : SInt;   // Speed 0–100 ( 0 = Stop, 100 = max speed), negative sign reverses the turning direction
   "IMC84MotorTargetSpeedRD -G1.4.2" AT %QB66 : SInt;   // Speed 0–100 ( 0 = Stop, 100 = max speed), negative sign reverses the turning direction
   "IMC84MotorTargetSpeedRD -G1.4.1" AT %QB67 : SInt;   // Speed 0–100 ( 0 = Stop, 100 = max speed), negative sign reverses the turning direction
   "IMC84MotorTargetSpeedRD_G1.3.1" AT %QB68 : SInt;   // Speed 0–100 ( 0 = Stop, 100 = max speed), negative sign reverses the turning direction
END_VAR

VAR_GLOBAL   // PLC tag table "BarcodeReader_DP1"
   "DP1-TriggerEnable" AT %Q81.0 : Bool;
   "DP1-Trigger" AT %Q81.1 : Bool;
   "DP1-TriggerReady" AT %I87.0 : Bool;
   "DP1-TriggerAck" AT %I87.1 : Bool;
   "DP1-Acquiring" AT %I87.2 : Bool;
   "DP1-MissedAcq" AT %I87.3 : Bool;
   "DP1-TriggerID" AT %IW88 : Word;
   "DP1-BufferResultsEnable" AT %Q82.0 : Bool;
   "DP1-ResultsAck" AT %Q82.1 : Bool;
   "DP1-Decoding" AT %I90.0 : Bool;
   "DP1-Decode Complete" AT %I90.1 : Bool;
   "DP1-Results Buffer Overrun" AT %I90.2 : Bool;
   "DP1-Results Available" AT %I90.3 : Bool;
   "DP1-General Fault" AT %I90.7 : Bool;
   "DP1-Train Code" AT %Q83.0 : Bool;
   "DP1-Train Match String" AT %Q83.1 : Bool;
   "DP1-Train Focus" AT %Q83.2 : Bool;
   "DP1-Train Brightness" AT %Q83.3 : Bool;
   "DP1-Untrain" AT %Q83.4 : Bool;
   "DP1-Execute DMCC" AT %Q83.6 : Bool;
   "DP1-Set Match String" AT %Q83.7 : Bool;
   "DP1-Train Code Ack" AT %I91.0 : Bool;
   "DP1-Train Match String Ack" AT %I91.1 : Bool;
   "DP1-Train Focus Ack" AT %I91.2 : Bool;
   "DP1-Train Brightness Ack" AT %I91.3 : Bool;
   "DP1-Untrain Ack" AT %I91.4 : Bool;
   "DP1-Execute DMCC Ack" AT %I91.6 : Bool;
   "DP1-Set Match String Ack" AT %I91.7 : Bool;
   "DP1-UserData Option" AT %QW84 : Word;
   "DP1-UserData Length" AT %QW86 : Word;
   "DP1-UserData[0]" AT %QB88 : Byte;
   "DP1-UserData[1]" AT %QB89 : Byte;
   "DP1-UserData[2]" AT %QB90 : Byte;
   "DP1-UserData[3]" AT %QB91 : Byte;
   "DP1-UserData[4]" AT %QB92 : Byte;
   "DP1-UserData[5]" AT %QB93 : Byte;
   "DP1-UserData[6]" AT %QB94 : Byte;
   "DP1-UserData[7]" AT %QB95 : Byte;
   "DP1-UserData[8]" AT %QB96 : Byte;
   "DP1-UserData[9]" AT %QB97 : Byte;
   "DP1-UserData[10]" AT %QB98 : Byte;
   "DP1-UserData[11]" AT %QB99 : Byte;
   "DP1-UserData[12]" AT %QB100 : Byte;
   "DP1-UserData[13]" AT %QB101 : Byte;
   "DP1-UserData[14]" AT %QB102 : Byte;
   "DP1-UserData[15]" AT %QB103 : Byte;
   "DP1-ResultID" AT %IW92 : Word;
   "DP1-Result Code" AT %IW95 : Word;
   "DP1-Read / No Read" AT %I95.0 : Bool;
   "DP1-Validated / Not Validated" AT %I95.1 : Bool;
   "DP1-Verified / Not Verified" AT %I95.2 : Bool;
   "DP1-Acquisition Trigger Overrun" AT %I95.3 : Bool;
   "DP1-Acquisition Buffer Overflow" AT %I95.4 : Bool;
   "DP1-Result Extended" AT %IW96 : Word;
   "DP1-Result Length" AT %IW98 : Word;
   "DP1-InspectionResults[0]" AT %IB100 : Byte;
   "DP1-InspectionResults[1]" AT %IB101 : Byte;
   "DP1-InspectionResults[2]" AT %IB102 : Byte;
   "DP1-InspectionResults[3]" AT %IB103 : Byte;
   "DP1-InspectionResults[4]" AT %IB104 : Byte;
   "DP1-InspectionResults[5]" AT %IB105 : Byte;
   "DP1-InspectionResults[6]" AT %IB106 : Byte;
   "DP1-InspectionResults[7]" AT %IB107 : Byte;
   "DP1-InspectionResults[8]" AT %IB108 : Byte;
   "DP1-InspectionResults[9]" AT %IB109 : Byte;
   "DP1-InspectionResults[10]" AT %IB110 : Byte;
   "DP1-InspectionResults[11]" AT %IB111 : Byte;
   "DP1-InspectionResults[12]" AT %IB112 : Byte;
   "DP1-InspectionResults[13]" AT %IB113 : Byte;
   "DP1-InspectionResults[14]" AT %IB114 : Byte;
   "DP1-InspectionResults[15]" AT %IB115 : Byte;
   "Result data_DP1" AT %I100.0 : "Global.BarCode";
   UserData_DP1 AT %Q88.0 : "Global.BarCode";
   ContinousGetResults_DP1 AT %M110.1 : Bool;
   TrainFocus_DP1 AT %M110.2 : Bool;
END_VAR

VAR_GLOBAL   // PLC tag table "BarcodeReader_DP2"
   "DP2-TriggerEnable" AT %Q152.0 : Bool;
   "DP2-Trigger" AT %Q152.1 : Bool;
   "DP2-TriggerReady" AT %I164.0 : Bool;
   "DP2-TriggerAck" AT %I164.1 : Bool;
   "DP2-Acquiring" AT %I164.2 : Bool;
   "DP2-MissedAcq" AT %I164.3 : Bool;
   "DP2-TriggerID" AT %IW165 : Word;
   "DP2-BufferResultsEnable" AT %Q153.0 : Bool;
   "DP2-ResultsAck" AT %Q153.1 : Bool;
   "DP2-Decoding" AT %I167.0 : Bool;
   "DP2-Decode Complete" AT %I167.1 : Bool;
   "DP2-Results Buffer Overrun" AT %I167.2 : Bool;
   "DP2-Results Available" AT %I167.3 : Bool;
   "DP2-General Fault" AT %I167.7 : Bool;
   "DP2-Train Code" AT %Q154.0 : Bool;
   "DP2-Train Match String" AT %Q154.1 : Bool;
   "DP2-Train Focus" AT %Q154.2 : Bool;
   "DP2-Train Brightness" AT %Q154.3 : Bool;
   "DP2-Untrain" AT %Q154.4 : Bool;
   "DP2-Execute DMCC" AT %Q154.6 : Bool;
   "DP2-Set Match String" AT %Q154.7 : Bool;
   "DP2-Train Code Ack" AT %I168.0 : Bool;
   "DP2-Train Match String Ack" AT %I168.1 : Bool;
   "DP2-Train Focus Ack" AT %I168.2 : Bool;
   "DP2-Train Brightness Ack" AT %I168.3 : Bool;
   "DP2-Untrain Ack" AT %I168.4 : Bool;
   "DP2-Execute DMCC Ack" AT %I168.6 : Bool;
   "DP2-Set Match String Ack" AT %I168.7 : Bool;
   "DP2-UserData Option" AT %QW155 : Word;
   "DP2-UserData Length" AT %QW157 : Word;
   "DP2-UserData[0]" AT %QB159 : Byte;
   "DP2-UserData[1]" AT %QB160 : Byte;
   "DP2-UserData[2]" AT %QB161 : Byte;
   "DP2-UserData[3]" AT %QB162 : Byte;
   "DP2-UserData[4]" AT %QB163 : Byte;
   "DP2-UserData[5]" AT %QB164 : Byte;
   "DP2-UserData[6]" AT %QB165 : Byte;
   "DP2-UserData[7]" AT %QB166 : Byte;
   "DP2-UserData[8]" AT %QB167 : Byte;
   "DP2-UserData[9]" AT %QB168 : Byte;
   "DP2-UserData[10]" AT %QB169 : Byte;
   "DP2-UserData[11]" AT %QB170 : Byte;
   "DP2-UserData[12]" AT %QB171 : Byte;
   "DP2-UserData[13]" AT %QB172 : Byte;
   "DP2-UserData[14]" AT %QB173 : Byte;
   "DP2-UserData[15]" AT %QB174 : Byte;
   "DP2-ResultID" AT %IW169 : Word;
   "DP2-Result Code" AT %IW172 : Word;
   "DP2-Read / No Read" AT %I172.0 : Bool;
   "DP2-Validated / Not Validated" AT %I172.1 : Bool;
   "DP2-Verified / Not Verified" AT %I172.2 : Bool;
   "DP2-Acquisition Trigger Overrun" AT %I172.3 : Bool;
   "DP2-Acquisition Buffer Overflow" AT %I172.4 : Bool;
   "DP2-Result Extended" AT %IW173 : Word;
   "DP2-Result Length" AT %IW175 : Word;
   "DP2-InspectionResults[0]" AT %IB177 : Byte;
   "DP2-InspectionResults[1]" AT %IB178 : Byte;
   "DP2-InspectionResults[2]" AT %IB179 : Byte;
   "DP2-InspectionResults[3]" AT %IB180 : Byte;
   "DP2-InspectionResults[4]" AT %IB181 : Byte;
   "DP2-InspectionResults[5]" AT %IB182 : Byte;
   "DP2-InspectionResults[6]" AT %IB183 : Byte;
   "DP2-InspectionResults[7]" AT %IB184 : Byte;
   "DP2-InspectionResults[8]" AT %IB185 : Byte;
   "DP2-InspectionResults[9]" AT %IB186 : Byte;
   "DP2-InspectionResults[10]" AT %IB187 : Byte;
   "DP2-InspectionResults[11]" AT %IB188 : Byte;
   "DP2-InspectionResults[12]" AT %IB189 : Byte;
   "DP2-InspectionResults[13]" AT %IB190 : Byte;
   "DP2-InspectionResults[14]" AT %IB191 : Byte;
   "DP2-InspectionResults[15]" AT %IB192 : Byte;
   "Result data_DP2" AT %I177.0 : "Global.BarCode";
   UserData_DP2 AT %Q159.0 : "Global.BarCode";
   ContinousGetResults_DP2 AT %M210.1 : Bool;
   TrainFocus_DP2 AT %M210.2 : Bool;
END_VAR

VAR_GLOBAL   // PLC tag table "BarcodeReader_DP3"
   "DP3-TriggerEnable" AT %Q223.0 : Bool;
   "DP3-Trigger" AT %Q223.1 : Bool;
   "DP3-TriggerReady" AT %I241.0 : Bool;
   "DP3-TriggerAck" AT %I241.1 : Bool;
   "DP3-Acquiring" AT %I241.2 : Bool;
   "DP3-MissedAcq" AT %I241.3 : Bool;
   "DP3-TriggerID" AT %IW242 : Word;
   "DP3-BufferResultsEnable" AT %Q224.0 : Bool;
   "DP3-ResultsAck" AT %Q224.1 : Bool;
   "DP3-Decoding" AT %I244.0 : Bool;
   "DP3-Decode Complete" AT %I244.1 : Bool;
   "DP3-Results Buffer Overrun" AT %I244.2 : Bool;
   "DP3-Results Available" AT %I244.3 : Bool;
   "DP3-General Fault" AT %I244.7 : Bool;
   "DP3-Train Code" AT %Q225.0 : Bool;
   "DP3-Train Match String" AT %Q225.1 : Bool;
   "DP3-Train Focus" AT %Q225.2 : Bool;
   "DP3-Train Brightness" AT %Q225.3 : Bool;
   "DP3-Untrain" AT %Q225.4 : Bool;
   "DP3-Execute DMCC" AT %Q225.6 : Bool;
   "DP3-Set Match String" AT %Q225.7 : Bool;
   "DP3-Train Code Ack" AT %I245.0 : Bool;
   "DP3-Train Match String Ack" AT %I245.1 : Bool;
   "DP3-Train Focus Ack" AT %I245.2 : Bool;
   "DP3-Train Brightness Ack" AT %I245.3 : Bool;
   "DP3-Untrain Ack" AT %I245.4 : Bool;
   "DP3-Execute DMCC Ack" AT %I245.6 : Bool;
   "DP3-Set Match String Ack" AT %I245.7 : Bool;
   "DP3-UserData Option" AT %QW226 : Word;
   "DP3-UserData Length" AT %QW228 : Word;
   "DP3-UserData[0]" AT %QB230 : Byte;
   "DP3-UserData[1]" AT %QB231 : Byte;
   "DP3-UserData[2]" AT %QB232 : Byte;
   "DP3-UserData[3]" AT %QB233 : Byte;
   "DP3-UserData[4]" AT %QB234 : Byte;
   "DP3-UserData[5]" AT %QB235 : Byte;
   "DP3-UserData[6]" AT %QB236 : Byte;
   "DP3-UserData[7]" AT %QB237 : Byte;
   "DP3-UserData[8]" AT %QB238 : Byte;
   "DP3-UserData[9]" AT %QB239 : Byte;
   "DP3-UserData[10]" AT %QB240 : Byte;
   "DP3-UserData[11]" AT %QB241 : Byte;
   "DP3-UserData[12]" AT %QB242 : Byte;
   "DP3-UserData[13]" AT %QB243 : Byte;
   "DP3-UserData[14]" AT %QB244 : Byte;
   "DP3-UserData[15]" AT %QB245 : Byte;
   "DP3-ResultID" AT %IW246 : Word;
   "DP3-Result Code" AT %IW249 : Word;
   "DP3-Read / No Read" AT %I249.0 : Bool;
   "DP3-Validated / Not Validated" AT %I249.1 : Bool;
   "DP3-Verified / Not Verified" AT %I249.2 : Bool;
   "DP3-Acquisition Trigger Overrun" AT %I249.3 : Bool;
   "DP3-Acquisition Buffer Overflow" AT %I249.4 : Bool;
   "DP3-Result Extended" AT %IW250 : Word;
   "DP3-Result Length" AT %IW252 : Word;
   "DP3-InspectionResults[0]" AT %IB254 : Byte;
   "DP3-InspectionResults[1]" AT %IB255 : Byte;
   "DP3-InspectionResults[2]" AT %IB256 : Byte;
   "DP3-InspectionResults[3]" AT %IB257 : Byte;
   "DP3-InspectionResults[4]" AT %IB258 : Byte;
   "DP3-InspectionResults[5]" AT %IB259 : Byte;
   "DP3-InspectionResults[6]" AT %IB260 : Byte;
   "DP3-InspectionResults[7]" AT %IB261 : Byte;
   "DP3-InspectionResults[8]" AT %IB262 : Byte;
   "DP3-InspectionResults[9]" AT %IB263 : Byte;
   "DP3-InspectionResults[10]" AT %IB264 : Byte;
   "DP3-InspectionResults[11]" AT %IB265 : Byte;
   "DP3-InspectionResults[12]" AT %IB266 : Byte;
   "DP3-InspectionResults[13]" AT %IB267 : Byte;
   "DP3-InspectionResults[14]" AT %IB268 : Byte;
   "DP3-InspectionResults[15]" AT %IB269 : Byte;
   "Result data_DP3" AT %I254.0 : "Global.BarCode";
   UserData_DP3 AT %Q230.0 : "Global.BarCode";
   ContinousGetResults_DP3 AT %M310.1 : Bool;
   TrainFocus_DP3 AT %M310.2 : Bool;
END_VAR

VAR_GLOBAL   // PLC tag table "BarcodeReader_DP4"
   "DP4-TriggerEnable" AT %Q294.0 : Bool;
   "DP4-Trigger" AT %Q294.1 : Bool;
   "DP4-TriggerReady" AT %I318.0 : Bool;
   "DP4-TriggerAck" AT %I318.1 : Bool;
   "DP4-Acquiring" AT %I318.2 : Bool;
   "DP4-MissedAcq" AT %I318.3 : Bool;
   "DP4-TriggerID" AT %IW319 : Word;
   "DP4-BufferResultsEnable" AT %Q295.0 : Bool;
   "DP4-ResultsAck" AT %Q295.1 : Bool;
   "DP4-Decoding" AT %I321.0 : Bool;
   "DP4-Decode Complete" AT %I321.1 : Bool;
   "DP4-Results Buffer Overrun" AT %I321.2 : Bool;
   "DP4-Results Available" AT %I321.3 : Bool;
   "DP4-General Fault" AT %I321.7 : Bool;
   "DP4-Train Code" AT %Q296.0 : Bool;
   "DP4-Train Match String" AT %Q296.1 : Bool;
   "DP4-Train Focus" AT %Q296.2 : Bool;
   "DP4-Train Brightness" AT %Q296.3 : Bool;
   "DP4-Untrain" AT %Q296.4 : Bool;
   "DP4-Execute DMCC" AT %Q296.6 : Bool;
   "DP4-Set Match String" AT %Q296.7 : Bool;
   "DP4-Train Code Ack" AT %I322.0 : Bool;
   "DP4-Train Match String Ack" AT %I322.1 : Bool;
   "DP4-Train Focus Ack" AT %I322.2 : Bool;
   "DP4-Train Brightness Ack" AT %I322.3 : Bool;
   "DP4-Untrain Ack" AT %I322.4 : Bool;
   "DP4-Execute DMCC Ack" AT %I322.6 : Bool;
   "DP4-Set Match String Ack" AT %I322.7 : Bool;
   "DP4-UserData Option" AT %QW297 : Word;
   "DP4-UserData Length" AT %QW299 : Word;
   "DP4-UserData[0]" AT %QB301 : Byte;
   "DP4-UserData[1]" AT %QB302 : Byte;
   "DP4-UserData[2]" AT %QB303 : Byte;
   "DP4-UserData[7]" AT %QB308 : Byte;
   "DP4-UserData[8]" AT %QB309 : Byte;
   "DP4-UserData[14]" AT %QB315 : Byte;
   "DP4-UserData[15]" AT %QB316 : Byte;
   "DP4-ResultID" AT %IW323 : Word;
   "DP4-Result Code" AT %IW326 : Word;
   "DP4-Read / No Read" AT %I326.0 : Bool;
   "DP4-Validated / Not Validated" AT %I326.1 : Bool;
   "DP4-Verified / Not Verified" AT %I326.2 : Bool;
   "DP4-Acquisition Trigger Overrun" AT %I326.3 : Bool;
   "DP4-Acquisition Buffer Overflow" AT %I326.4 : Bool;
   "DP4-Result Extended" AT %IW327 : Word;
   "DP4-InspectionResults[10]" AT %IB341 : Byte;
   "DP4-InspectionResults[11]" AT %IB342 : Byte;
   "DP4-InspectionResults[12]" AT %IB343 : Byte;
   "DP4-InspectionResults[13]" AT %IB344 : Byte;
   "DP4-InspectionResults[14]" AT %IB345 : Byte;
   "DP4-InspectionResults[15]" AT %IB346 : Byte;
   ContinousGetResults_DP4 AT %M10.1 : Bool;
   TrainFocus_DP4 AT %M10.2 : Bool;
   "DP4-Result Length" AT %IW329 : Word;
   "DP4-InspectionResults[0]" AT %IB331 : Byte;
   "DP4-InspectionResults[1]" AT %IB332 : Byte;
   "DP4-InspectionResults[2]" AT %IB333 : Byte;
   "DP4-InspectionResults[3]" AT %IB334 : Byte;
   "DP4-InspectionResults[4]" AT %IB335 : Byte;
   "DP4-InspectionResults[5]" AT %IB336 : Byte;
   "DP4-InspectionResults[6]" AT %IB337 : Byte;
   "DP4-InspectionResults[7]" AT %IB338 : Byte;
   "DP4-InspectionResults[8]" AT %IB339 : Byte;
   "DP4-InspectionResults[9]" AT %IB340 : Byte;
   "Result data_DP4" AT %I331.0 : "Global.BarCode";
   "DP4-UserData[3]" AT %QB304 : Byte;
   "DP4-UserData[4]" AT %QB305 : Byte;
   "DP4-UserData[5]" AT %QB306 : Byte;
   "DP4-UserData[6]" AT %QB307 : Byte;
   "DP4-UserData[9]" AT %QB310 : Byte;
   "DP4-UserData[10]" AT %QB311 : Byte;
   "DP4-UserData[11]" AT %QB312 : Byte;
   "DP4-UserData[12]" AT %QB313 : Byte;
   "DP4-UserData[13]" AT %QB314 : Byte;
   UserData_DP4 AT %Q301.0 : "Global.BarCode";
END_VAR

VAR_GLOBAL   // PLC tag table "IMC88"
   IMC88Sensor_1 AT %I727.0 : Bool;   // High = Sensor active (input type and polarity can be configured)
   IMC88Sensor_2 AT %I727.1 : Bool;   // High = Sensor active (input type and polarity can be configured)
   IMC88Sensor_3 AT %I727.2 : Bool;   // High = Sensor active (input type and polarity can be configured)
   IMC88Sensor_4 AT %I727.3 : Bool;   // High = Sensor active (input type and polarity can be configured)
   IMC88Sensor_5 AT %I727.4 : Bool;
   IMC88Sensor_6 AT %I727.5 : Bool;
   IMC88Sensor_7 AT %I727.6 : Bool;
   IMC88Sensor_8 AT %I727.7 : Bool;
   IMC88IO1 AT %I728.0 : Bool;   // Digital I/O PLC Input PLC Output
   IMC88IO2 AT %I728.1 : Bool;   // Digital I/O PLC Input PLC Output
   IMC88IO3 AT %I728.2 : Bool;   // Digital I/O PLC Input PLC Output
   IMC88IO4 AT %I728.3 : Bool;   // Digital I/O PLC Input PLC Output
   IMC88IO5 AT %I728.4 : Bool;
   IMC88IO6 AT %I728.5 : Bool;
   IMC88IO7 AT %I728.6 : Bool;
   IMC88IO8 AT %I728.7 : Bool;
   "IMC88MotorStateErrorRD -G1.7.4" AT %I729.0 : Bool;   // High = Motor Error; Low = Motor OK
   "IMC88MotorStateErrorRD -G1.7.3" AT %I729.1 : Bool;   // High = Motor Error; Low = Motor OK
   "IMC88MotorStateErrorRD -G1.7.2" AT %I729.2 : Bool;   // High = Motor Error; Low = Motor OK
   "IMC88MotorStateErrorRD -4" AT %I729.3 : Bool;   // High = Motor Error; Low = Motor OK
   "IMC88MotorStateSpeedRD -G1.7.4" AT %IB730 : SInt;   // Speed 0–100 ( 0 = Stop, 100 = max speed), negative sign reverses the turning direction
   "IMC88MotorStateSpeedRD -G1.7.3" AT %IB731 : SInt;   // Speed 0–100 ( 0 = Stop, 100 = max speed), negative sign reverses the turning direction
   "IMC88MotorStateSpeedRD -G1.7.2" AT %IB732 : SInt;   // Speed 0–100 ( 0 = Stop, 100 = max speed), negative sign reverses the turning direction
   "IMC88MotorStateSpeedRD -4" AT %IB733 : SInt;   // Speed 0–100 ( 0 = Stop, 100 = max speed), negative sign reverses the turning direction
   "IMC88MotorCurrentRD -G1.7.4" AT %IW735 : Int;   // Average current in mA
   "IMC88MotorCurrentRD -G1.7.3" AT %IW737 : Int;   // Average current in mA
   "IMC88MotorCurrentRD -G1.7.2" AT %IW739 : Int;   // Average current in mA
   "IMC88MotorCurrentRD -4" AT %IW741 : Int;   // Average current in mA
   "IMC88Voltage(MotorPower)" AT %IW743 : Int;   // Voltage „Motor Power“ in mV
   "IMC88Voltage(Sensors)" AT %IW745 : Int;   // Voltage „Power Logic + Sensors“ in mV
   IMC88Temperature AT %IW747 : Int;   // Temperature in 0,1 C
   IMC88SystemUpTime AT %ID749 : DInt;   // Operating time in seconds since the last start/restart
   "IMC88DigitalOutputRD -G1.7.4" AT %Q535.0 : Bool;
   "IMC88DigitalOutputRD -G1.7.3" AT %Q535.1 : Bool;
   "IMC88DigitalOutputRD -G1.7.2" AT %Q535.2 : Bool;
   "IMC88DigitalOutputRD -4" AT %Q535.3 : Bool;
   "IMC88MotorTargetSpeedRD -G1.7.4" AT %QB536 : SInt;   // Speed 0–100 ( 0 = Stop, 100 = max speed), negative sign reverses the turning direction
   "IMC88MotorTargetSpeedRD -G1.7.3" AT %QB537 : SInt;   // Speed 0–100 ( 0 = Stop, 100 = max speed), negative sign reverses the turning direction
   "IMC88MotorTargetSpeedRD -G1.7.2" AT %QB538 : SInt;   // Speed 0–100 ( 0 = Stop, 100 = max speed), negative sign reverses the turning direction
   "IMC88MotorTargetSpeedRD -4" AT %QB539 : SInt;   // Speed 0–100 ( 0 = Stop, 100 = max speed), negative sign reverses the turning direction
END_VAR

TYPE "BarCode"
// stored: Namespace Global
   STRUCT
      "Result Data" : Array[0..63] of Byte;
   END_STRUCT;
END_TYPE

TYPE "ConveyorParameters"
// stored: Access Published, Namespace Global
   STRUCT
      StartUpTime : Time := T#0S;
      SensorFilterTime : Array[1..2] of Time;
      SensorBlockageTime : Time := T#5S;
      EnergySaveTime : Time := T#3s;
      ConvOccTime : Time := T#1000ms;
   END_STRUCT;
   // SensorFilterTime[1..2] := T#10ms;
END_TYPE

TYPE "ConveyorStatus"
// stored: Access Published, Namespace Global
   STRUCT
      Blockage : Bool;
      xReserved_2 : Bool;
      xReserved_3 : Bool;
      xReserved_4 : Bool;
      xReserved_5 : Bool;
      xReserved_6 : Bool;
      xReserved_7 : Bool;
      xReserved_8 : Bool;
      ON : Bool;
      ReadytoRun : Bool;
      Occupied : Bool;
      Running : Bool;
      Fault : Bool;
      Estop : Bool;
      Manual : Bool;
      Stop : Bool;
   END_STRUCT;
END_TYPE

TYPE "Fault"
// stored: Access Published, Namespace Global
   STRUCT
      Motor_Error : Bool;
      Sensor_Blockage : Bool;
   END_STRUCT;
END_TYPE

TYPE "GetDiag"
// stored: Access Published, Namespace Global
   STRUCT
      DiagMode : UInt := 1;
      CommID : HW_ANY;
      ReturnValue : Int;
      CountDiagDetail : UInt;
      MyDiag : DIS;
   END_STRUCT;
END_TYPE

TYPE "ItemDir"
// stored: Access Published, Namespace Global
   STRUCT
      Straight : Bool;
      toRight : Bool;
      toLeft : Bool;
   END_STRUCT;
END_TYPE

TYPE "ManualInputs"
// stored: Access Published, Namespace Global
   STRUCT
      ManualEnable : Bool;
      Run : Struct
         Forward : Bool;
         Reverse : Bool;
      END_STRUCT;
   END_STRUCT;
END_TYPE

TYPE "S300Manual"
// stored: Access Published, Namespace Global
   STRUCT
      GoUp : Bool;
      GoStraight : Bool;
      GoLeft : Bool;
      GoRight : Bool;
   END_STRUCT;
END_TYPE

TYPE "SystemSSR"
// stored: Access Published, Namespace Global
   STRUCT
      StartSystem : Bool;   // Start the system
      StopSystem : Bool;   // Stop the system
      ResetSystem : Bool;   // Reset the system
   END_STRUCT;
END_TYPE

TYPE "TrackingData"
// stored: Access Published, Namespace Global
   STRUCT
      Barcode : String;
      ResponseCode : UInt;
      HeightLimit : Bool;
      ActualWeight : Struct
         inRealValue : Real;
         inStringFormat : String;
      END_STRUCT;
      EXIT_1_ : Array[1..1] of Bool;
      EXIT_2_ : Array[1..6] of Bool;
      ToteDir : "Global.ItemDir";
   END_STRUCT;
END_TYPE

TYPE "MABS_Parameters"
// stored: Namespace LineA1
   STRUCT
      StartUpTime : Time := T#5S;
      CrossSensorFilterTime : Array[1..2] of Time;
      SensorBlockageTime : Time := T#5S;
      EnergySaveTime : Time := T#4s;
   END_STRUCT;
END_TYPE

TYPE "setTransferTimer"
// stored: Access Published, Namespace LineC1
   STRUCT
      setTransferTimer : Array[1..2] of Time;
   END_STRUCT;
END_TYPE

TYPE "ConveyorParameters_TransferUnit"
// stored: Access Published, Namespace Global
   STRUCT
      StartUpTime : Time := T#0S;
      SensorFilterTime : Array[1..2] of Time;
      FrontSensorFilterTime : Array[1..2] of Time;
      "Left/RightSensorFilterTime" : Array[1..2] of Time;
      EndsensorFilterTime : Array[1..2] of Time;
      SensorBlockageTime : Time := T#5S;
      EnergySaveTime : Time := T#3s;
      ConvOccTime : Time := T#1000ms;
   END_STRUCT;
   // SensorFilterTime[1..2] := T#10ms;
   // FrontSensorFilterTime[1..2] := T#10ms;
   // "Left/RightSensorFilterTime"[1..2] := T#10ms;
END_TYPE

TYPE "EsopZone"
// stored: Access Published, Namespace Global
   STRUCT
      "1" : Bool;
      "2" : Bool;
   END_STRUCT;
END_TYPE

TYPE "S300ForceMode"
// stored: Access Published, Namespace Global
   STRUCT
      BeltDir : Bool;
      RollerDir : Bool;
   END_STRUCT;
END_TYPE

TYPE "MABS"
// stored: Access Published, Namespace Global
   STRUCT
      Run_balls : Bool := false;   // Run transport balls
      Dir_balls : Bool := false;   // 0=forward; 1=backward
      Speed_balls : Int := 90;   // Based on preset speed setting. 60/70/80/90 m/min.
      Switch_left_angle : Int := 45;   // Angle for left transportation 30/180°
      Switch_right_angle : Int := 45;   // Angle for right transportation 30/180°
      Switch_left_to_st_offset : Int := 0;   // Offset angle for straight position from left -8/+10°
      Switch_right_to_st_offset : Int := 0;   // Offset angle for straight position from right -8/+10°
      Init_offset : Int := 0;   // Offset angle for initial position -8/+10°
      Switch_left : Bool := false;   // Swing to left transport direction
      Switch_right : Bool := false;   // Swing to right transport direction
      Switch_left_to_st : Bool := false;   // Swing to straight transport direction CW
      Switch_right_to_st : Bool := false;   // Swing to straight transport direction CCW
      EMS : Bool := false;   // Inhib controls and reset MABS initialisation
      Init : Bool := false;   // Run MABS initialisation sequence (if not done)
      Init_done : Bool := false;   // MABS initialisation sequence done
      Ready : Bool := false;   // MABS no error, initialisation done, communication OK
      Init_sensor : Bool := false;   // MABS straight position sensor
      Left_Pos_reach : Bool := false;   // MABS transport balls in left position
      Right_Pos_reach : Bool := false;   // MABS transport balls in right position
      Straight_Pos_reach : Bool := false;   // MABS transport balls in straight position
      Error_motA : Bool := false;   // Hardware error motor A
      Error_motB : Bool := false;   // Hardware error motor B
      Error_timeout_sw : Bool := false;   // Swing motor timeout
      Error_com : Bool := false;   // Communication error (life bit, 5s delayed)
      Error : Bool := false;   // Error synthesis
      Reset_error : Bool := false;   // Reset all errors
      Timeout_val : Time := T#10s;   // Swing timeout value
      HMI_sts : UInt := 0;   // Sts word for HMI (0=Off; 1=Running; 2=Init requested; 4=Error )
   END_STRUCT;
END_TYPE

TYPE "MABS_ManIn"
// stored: Access Published, Namespace Global
   STRUCT
      RunBalls : Bool;
      Switch : Struct
         ToLeft : Bool;
         ToRight : Bool;
         left_to_st : Bool;
         right_to_st : Bool;
      END_STRUCT;
   END_STRUCT;
END_TYPE

TYPE "MABS_Setpoint"
// stored: Access Published, Namespace Global
   STRUCT
      ChangeBallsDirection : Bool;   // 0=forward; 1=backward
      Speed_balls : Int := 0;   // Based on preset speed setting. 60/70/80/90 m/min.
      Init_offset : Int;   // Offset angle for initial position -8/+10°
   END_STRUCT;
END_TYPE

TYPE "IB_P01_02_03_in_64bytes_struct"
// stored: Access Published, Namespace Global
   STRUCT
      Reserved : Byte;
      Sens_A : Bool;
      Sens_B : Bool;
      Sens_A_alrm : Bool;
      Sens_B_alrm : Bool;
      Motor_state_A : Bool;
      Motor_state_B : Bool;
      Reserved_1 : Bool;
      Reserved_2 : Bool;
      Fuse_err_A : Bool;
      Back_EMF_err_A : Bool;
      Thermal_err_mot_A : Bool;
      Thermal_err_ctrl_A : Bool;
      Lock_err_A : Bool;
      Unconnected_err_A : Bool;
      Reserved_3 : Bool;
      Reserved_4 : Bool;
      Fuse_err_B : Bool;
      Back_EMF_err_B : Bool;
      Thermal_err_mot_B : Bool;
      Thermal_err_ctrl_B : Bool;
      Lock_err_B : Bool;
      Unconnected_err_B : Bool;
      Reserved_5 : Bool;
      Reserved_6 : Bool;
      Digital_in_1 : Bool;   // NA for IB-P03
      Digital_in_2 : Bool;   // NA for IB-P03
      Digital_in_3 : Bool;   // NA for IB-P03
      Digital_in_4 : Bool;   // NA for IB-P03
      Reserved_7 : Bool;
      Reserved_8 : Bool;
      Reserved_9 : Bool;
      Reserved_10 : Bool;
      Register_Low_D0 : Byte;
      Register_High_D0 : Byte;
      Register_Low_D1 : Byte;
      Register_High_D1 : Byte;
      Register_Low_D2 : Byte;
      Register_High_D2 : Byte;
      Register_Low_D3 : Byte;
      Register_High_D3 : Byte;
      Register_Low_D4 : Byte;
      Register_High_D4 : Byte;
      Register_Low_D5 : Byte;
      Register_High_D5 : Byte;
      Register_Low_D6 : Byte;
      Register_High_D6 : Byte;
      Register_Low_D7 : Byte;
      Register_High_D7 : Byte;
      Register_Low_D8 : Byte;
      Register_High_D8 : Byte;
      Register_Low_D9 : Byte;
      Register_High_D9 : Byte;
      Register_Low_D10 : Byte;
      Register_High_D10 : Byte;
      Register_Low_D11 : Byte;
      Register_High_D11 : Byte;
      Register_Low_D12 : Byte;
      Register_High_D12 : Byte;
      Register_Low_D13 : Byte;
      Register_High_D13 : Byte;
      Register_Low_D14 : Byte;
      Register_High_D14 : Byte;
      Register_Low_D15 : Byte;
      Register_High_D15 : Byte;
      Life_time_mot_A_LL : Byte;
      Life_time_mot_A_LH : Byte;
      Life_time_mot_A_HL : Byte;
      Life_time_mot_A_HH : Byte;
      Life_time_mot_B_LL : Byte;
      Life_time_mot_B_LH : Byte;
      Life_time_mot_B_HL : Byte;
      Life_time_mot_B_HH : Byte;
      Current_mot_A : Byte;
      Current_mot_B : Byte;
      Voltage_mot_A : Byte;
      Voltage_mot_B : Byte;
      Reserved_11 : Array[0..13] of Byte;
   END_STRUCT;
END_TYPE

TYPE "IB_P01_02_03_out_64bytes_struct"
// stored: Access Published, Namespace Global
   STRUCT
      Run_mot_A : Bool;
      Run_mot_B : Bool;
      Reserved_1 : Bool;
      Reserved_2 : Bool;
      Reserved_3 : Bool;
      Reserved_4 : Bool;
      Reserved_5 : Bool;
      Reserved_6 : Bool;
      Speed_1_A : Bool;
      Speed_2_A : Bool;
      Speed_3_A : Bool;
      Speed_4_A : Bool;
      Speed_1_B : Bool;
      Speed_2_B : Bool;
      Speed_3_B : Bool;
      Speed_4_B : Bool;
      Acc_A : Bool;
      Dec_A : Bool;
      Acc_B : Bool;
      Dec_B : Bool;
      Dir_A : Bool;
      Dir_B : Bool;
      Ack_err_A : Bool;
      Ack_err_B : Bool;
      Digital_out1 : Bool;   // NA for IB-P03
      Digital_out2 : Bool;   // NA for IB-P03
      Digital_out3 : Bool;   // NA for IB-P03
      Digital_out4 : Bool;   // NA for IB-P03
      Reserved_7 : Bool;
      Reserved_8 : Bool;
      Reserved_9 : Bool;
      Reserved_10 : Bool;
      Register_Low_D800 : Byte;
      Register_High_D800 : Byte;
      Register_Low_D801 : Byte;
      Register_High_D801 : Byte;
      Register_Low_D802 : Byte;
      Register_High_D802 : Byte;
      Register_Low_D803 : Byte;
      Register_High_D803 : Byte;
      Register_Low_D804 : Byte;
      Register_High_D804 : Byte;
      Register_Low_D805 : Byte;
      Register_High_D805 : Byte;
      Register_Low_D806 : Byte;
      Register_High_D806 : Byte;
      Register_Low_D807 : Byte;
      Register_High_D807 : Byte;
      Register_Low_D808 : Byte;
      Register_High_D808 : Byte;
      Register_Low_D809 : Byte;
      Register_High_D809 : Byte;
      Register_Low_D810 : Byte;
      Register_High_D810 : Byte;
      Register_Low_D811 : Byte;
      Register_High_D811 : Byte;
      Register_Low_D812 : Byte;
      Register_High_D812 : Byte;
      Register_Low_D813 : Byte;
      Register_High_D813 : Byte;
      Register_Low_D814 : Byte;
      Register_High_D814 : Byte;
      Register_Low_D815 : Byte;
      Register_High_D815 : Byte;
      Output_stop : Byte;
      Led_JAM_A : Bool;
      Led_JAM_B : Bool;
      Led_soft1_A : Bool;
      Led_soft1_B : Bool;
      Led_soft2_A : Bool;
      Led_soft2_B : Bool;
      Reserved_11 : Bool;
      Reserved_12 : Bool;
      Reserved_13 : Array[0..25] of Byte;
   END_STRUCT;
END_TYPE

TYPE "Log_Data_Byte_Decimal"
// stored: Namespace ProductionLine
   STRUCT
      DataType : Int;
      Representation : Int;
      RepreLength : Int;
      Reserve : Int;
      Data : Int;
   END_STRUCT;
END_TYPE

TYPE "Log_Data_Char"
// stored: Namespace ProductionLine
   STRUCT
      DataType : Byte;
      Representation : Byte;
      RepreLength : Byte;
      Reserve : Byte;
      Data : Char;
   END_STRUCT;
END_TYPE

TYPE "Log_Data_String20"
// stored: Namespace ProductionLine
   STRUCT
      DataType : Byte;
      Representation : Byte;
      RepreLength : Byte;
      Reserve : Byte;
      Data : String[20];
   END_STRUCT;
END_TYPE

TYPE "Log_LogMsg_Header"
// stored: Namespace ProductionLine
   STRUCT
      STX : Byte;
      SOH : Byte;
      MsgLength : Int;
      MsgType : Byte;
      Reserve : Byte;
      EventLevel : Byte;
      EventGroup : Byte;
      Timestamp : Date_And_Time;
      EventID : Int;
   END_STRUCT;
END_TYPE

TYPE "OPC_DestAssign"
// stored: Namespace ProductionLine
   STRUCT
      SourceSeq : Int;
      SourceNode : String[8];
      TotesID : String[10];
      WMSID : String[20];
      DestinationNode : String[8];
   END_STRUCT;
END_TYPE

TYPE "OPC_DestAssign_Ack"
// stored: Namespace ProductionLine
   STRUCT
      AckSeq : Int;
      SourceNode : String[8];
      TotesID : String[10];
      WMSID : String[20];
      Confirmation : String[1];
   END_STRUCT;
END_TYPE

TYPE "OPC_DestInfo"
// stored: Namespace ProductionLine
   STRUCT
      SourceSeq : Int;   // //Communication flag, described in the Request - Response tab
      DecisionPoint : String[30];   // // Machine/workstation code: - DP1,…, DP4
      Barcode : String[30];   // // Unique identification of scanned KLTs. For NoRead use ??????????
      InformationPoint : String[30];   // // Identification of the target location: - IP1...IP9
   END_STRUCT;
END_TYPE

TYPE "OPC_DestInfo_Ack"
// stored: Namespace ProductionLine
   STRUCT
      AckSeq : Int;   // //Communication flag, described in the Data tab
   END_STRUCT;
END_TYPE

TYPE "OPC_DestRequest_Ack"
// stored: Namespace ProductionLine
   STRUCT
      AckSeq : Int;   // //Communication flag, described in the Request - Response tab
      DecisionPoint : String[30];   // // Machine/workstation code:- DP1,…, DP4
      Barcode : String[30];   // // Unique identification of scanned KLTs. For NoRead use ??????????
      State : String[10];   // // Response status: - OK = task ready - NG (not good) = error
      Destination : String[30];   // Identification of the target location: - IP1...IP9
      ErrorReason : String[150];   // // Reason for error in case of status = NG.
   END_STRUCT;
END_TYPE

TYPE "OPC_DsetRequest"
// stored: Namespace ProductionLine
   STRUCT
      SourceSeq : Int;   // // Communication flag, described in the Request - Response tab
      DecisionPoint : String[30];   // // Machine/workstation code: - DP1,…, DP4
      Barcode : String[30];   // // Unique identification of scanned KLTs. For NoRead use ??????????
   END_STRUCT;
END_TYPE

TYPE "OPC_SegmentStatus"
// stored: Namespace ProductionLine
   STRUCT
      Segment : Struct
         FlowRackLoop : Int;
         FlowRackWorkplaceLeft : Int;
         FlowRackWorkplaceRight : Int;
         FragileLoop : Int;
      END_STRUCT;
   END_STRUCT;
END_TYPE

TYPE "OPC_SystStatus_Ack"
// stored: Namespace ProductionLine
   STRUCT
      AckSeq : Int;
   END_STRUCT;
END_TYPE

TYPE "OPC_SystemStatus"
// stored: Namespace ProductionLine
   STRUCT
      SourceSeq : Int;
   END_STRUCT;
END_TYPE

DATA_BLOCK "DB_Sync"   // DB3
{ S7_Optimized_Access := 'TRUE' }
// stored: MemoryReserve 100
   VAR
      memoryBit : Struct
         System_Byte : Byte;
         FirstScan : Bool;
         DiagStatusUpdate : Bool;
         AlwaysTRUE : Bool;
         AlwaysFALSE : Bool;
      END_STRUCT;
      ClockBit : Struct
         Clock_Byte : Byte;
         Clock_10Hz : Bool;
         Clock_5Hz : Bool;
         "Clock_2.5Hz" : Bool;
         Clock_2Hz : Bool;
         "Clock_1.25Hz" : Bool;
         Clock_1Hz : Bool;
         "Clock_0.625Hz" : Bool;
         "Clock_0.5Hz" : Bool;
      END_STRUCT;
      startbit : Bool;
      stopbit : Bool;
      resetbit : Bool;
   END_VAR
BEGIN
END_DATA_BLOCK

DATA_BLOCK "DB_SafetyStandard"   // DB20
// stored: Access Published, MemoryReserve 100
   VAR
      ToStandard : Struct
         EstopActive : Bool;
      END_STRUCT;
      PressReset : Bool;
      ToHMI : Struct
         "EstopPB -AS1.7.4 -SF09 -Zone2" : Bool;
         "EstopPB -AS1.12.3 -SF10 -Zone3" : Bool;
         "EstopPB -AS1.13.14 -SF11 -Zone3" : Bool;
         "EstopPB -AS1.55.2 -SF01 -Zone1" : Bool;
         "EstopPB -AS1.55.11 -SF02 -Zone1" : Bool;
         "EstopPB -AS1.55.18 -SF03 -Zone1" : Bool;
         "EstopPB -AS1.58.2 -SF04 -Zone1" : Bool;
         "EstopPB -AS1.58.11 -SF05 -Zone1" : Bool;
         "EstopPB -AS1.58.19 -SF06 -Zone1" : Bool;
         "EstopPB -AS1.5.9 -SF07 -Zone2" : Bool;
         "EstopPB -AS1.9.4 -SF08 -Zone2" : Bool;
         "EstopPB -MCC100 -402SF7" : Bool;
         "PhaseOK -MCC100" : Bool;
         "EstopPB -AS1.50.7 -SF21" : Bool;
         "EstopPB -AS1.50.24 -SF22" : Bool;
         "EstopPB -AS1.50.8 -SF23" : Bool;
         "EstopPB -BP1.2.42 -SF24" : Bool;
         "EstopPB -BP2.3.2 -SF25" : Bool;
         "EstopPB -BP1.14.3 -SF26" : Bool;
         "EstopPB -BP1.6.2 -SF27" : Bool;
         "EstopPB -MCC300 -402SF7" : Bool;
         "PhaseOK -MCC300" : Bool;
      END_STRUCT;
      holdAlarmOffTimer : TON_TIME;
      holdAlarmOff : Bool;
   END_VAR
BEGIN
END_DATA_BLOCK

DATA_BLOCK "DB_Global"   // DB23
// stored: Access Published, MemoryReserve 100, Namespace Global
   VAR
      Status : Struct
         Line : Struct
            A1 : Struct
               On : Array[_.gMinA1.._.gMaxA1] of Bool;
               ReadyToRun : Array[_.gMinA1.._.gMaxA1] of Bool;
               Occupied : Array[_.gMinA1.._.gMaxA1] of Bool;
               Running : Array[_.gMinA1.._.gMaxA1] of Bool;
               Fault : Array[_.gMinA1.._.gMaxA1] of Bool;
               Estop : Array[_.gMinA1.._.gMaxA1] of Bool;
               Manual : Array[_.gMinA1.._.gMaxA1] of Bool;
               Stop : Array[_.gMinA1.._.gMaxA1] of Bool;
               Blockage : Array[_.gMinA1.._.gMaxA1] of Bool;
            END_STRUCT;
            B1 : Struct
               On : Array[_.gMinB1.._.gMaxB1] of Bool;
               ReadyToRun : Array[_.gMinB1.._.gMaxB1] of Bool;
               Occupied : Array[_.gMinB1.._.gMaxB1] of Bool;
               Running : Array[_.gMinB1.._.gMaxB1] of Bool;
               Fault : Array[_.gMinB1.._.gMaxB1] of Bool;
               Estop : Array[_.gMinB1.._.gMaxB1] of Bool;
               Manual : Array[_.gMinB1.._.gMaxB1] of Bool;
               Stop : Array[_.gMinB1.._.gMaxB1] of Bool;
               Blockage : Array[_.gMinB1.._.gMaxB1] of Bool;
            END_STRUCT;
            C1 : Struct
               On : Array[_.gMinC1.._.gMaxC1] of Bool;
               ReadyToRun : Array[_.gMinC1.._.gMaxC1] of Bool;
               Occupied : Array[_.gMinC1.._.gMaxC1] of Bool;
               Running : Array[_.gMinC1.._.gMaxC1] of Bool;
               Fault : Array[_.gMinC1.._.gMaxC1] of Bool;
               Estop : Array[_.gMinC1.._.gMaxC1] of Bool;
               Manual : Array[_.gMinC1.._.gMaxC1] of Bool;
               Stop : Array[_.gMinC1.._.gMaxC1] of Bool;
               Blockage : Array[_.gMinC1.._.gMaxC1] of Bool;
            END_STRUCT;
            D1 : Struct
               On : Array[_.gMinD1.._.gMaxD1] of Bool;
               ReadyToRun : Array[_.gMinD1.._.gMaxD1] of Bool;
               Occupied : Array[_.gMinD1.._.gMaxD1] of Bool;
               Running : Array[_.gMinD1.._.gMaxD1] of Bool;
               Fault : Array[_.gMinD1.._.gMaxD1] of Bool;
               Estop : Array[_.gMinD1.._.gMaxD1] of Bool;
               Manual : Array[_.gMinD1.._.gMaxD1] of Bool;
               Stop : Array[_.gMinD1.._.gMaxD1] of Bool;
               Blockage : Array[_.gMinD1.._.gMaxD1] of Bool;
            END_STRUCT;
         END_STRUCT;
      END_STRUCT;
   END_VAR
BEGIN
   // Status.Line.A1.On[1001] : AS1.1.1
   // Status.Line.A1.On[1002] : AS1.1.2
   // Status.Line.A1.ReadyToRun[1001] : AS1.1.1
   // Status.Line.A1.ReadyToRun[1002] : AS1.1.2
   // Status.Line.A1.Occupied[1001] : AS1.1.1
   // Status.Line.A1.Occupied[1002] : AS1.1.2
   // Status.Line.A1.Running[1001] : AS1.1.1
   // Status.Line.A1.Running[1002] : AS1.1.2
   Status.Line.A1.Fault[1001] := 0;   // AS1.1.1
   Status.Line.A1.Fault[1002] := 0;   // AS1.1.2
   Status.Line.A1.Estop[1001] := 0;   // AS1.1.1
   Status.Line.A1.Estop[1002] := 0;   // AS1.1.2
   Status.Line.A1.Manual[1001] := 0;   // AS1.1.1
   Status.Line.A1.Manual[1002] := 0;   // AS1.1.2
   Status.Line.A1.Stop[1001] := 0;   // AS1.1.1
   Status.Line.A1.Stop[1002] := 0;   // AS1.1.2
   Status.Line.A1.Blockage[1001] := 0;   // AS1.1.1
   Status.Line.A1.Blockage[1002] := 0;   // AS1.1.2
   // Status.Line.C1.ReadyToRun[3001] : BP1.1.1
   // Status.Line.C1.ReadyToRun[3002] : BP1.1.2
   // Status.Line.C1.Occupied[3001] : BP1.1.1
   // Status.Line.C1.Occupied[3002] : BP1.1.2
   // Status.Line.C1.Running[3001] : BP1.1.1
   // Status.Line.C1.Running[3002] : BP1.1.2
   // Status.Line.C1.Fault[3001] : BP1.1.1
   // Status.Line.C1.Fault[3002] : BP1.1.2
   // Status.Line.C1.Estop[3001] : BP1.1.1
   // Status.Line.C1.Estop[3002] : BP1.1.2
   // Status.Line.C1.Manual[3001] : BP1.1.1
   // Status.Line.C1.Manual[3002] : BP1.1.2
   // Status.Line.C1.Stop[3001] : BP1.1.1
   // Status.Line.C1.Stop[3002] : BP1.1.2
   // Status.Line.C1.Blockage[3001] : BP1.1.1
   // Status.Line.C1.Blockage[3002] : BP1.1.2
END_DATA_BLOCK

DATA_BLOCK "DB_Temporary"   // DB40
// stored: MemoryReserve 100, Namespace EmptyLine
   VAR
      MABS1_In { ExternalAccessible := 'False'; ExternalVisible := 'False'; ExternalWritable := 'False'} : "Global.IB_P01_02_03_in_64bytes_struct";
      MABS1_Out { ExternalAccessible := 'False'; ExternalVisible := 'False'; ExternalWritable := 'False'} : "Global.IB_P01_02_03_out_64bytes_struct";
      MABS2_In { ExternalAccessible := 'False'; ExternalVisible := 'False'; ExternalWritable := 'False'} : "Global.IB_P01_02_03_in_64bytes_struct";
      MABS2_Out { ExternalAccessible := 'False'; ExternalVisible := 'False'; ExternalWritable := 'False'} : "Global.IB_P01_02_03_out_64bytes_struct";
   END_VAR
BEGIN
END_DATA_BLOCK

DATA_BLOCK "ToteDir"   // DB43
// stored: MemoryReserve 100, Namespace EmptyLine
   VAR
      Conveyor : Array[_."J1.6.1".._."J1.6.2"] of "Global.ItemDir";
   END_VAR
BEGIN
END_DATA_BLOCK

DATA_BLOCK "DB_SystemSSR"   // DB5
// stored: Access Published, MemoryReserve 100, Namespace Global
   VAR
      FromHMI : Struct
         Line : Struct
            A1 : "Global.SystemSSR";
            B1 { S7_SetPoint := 'True'} : "Global.SystemSSR";
            C1 { S7_SetPoint := 'True'} : "Global.SystemSSR";
            D1 { S7_SetPoint := 'True'} : "Global.SystemSSR";
         END_STRUCT;
      END_STRUCT;
      Line : Struct
         A1 : "Global.SystemSSR";
         B1 { S7_SetPoint := 'True'} : "Global.SystemSSR";
         C1 { S7_SetPoint := 'True'} : "Global.SystemSSR";
         D1 { S7_SetPoint := 'True'} : "Global.SystemSSR";
      END_STRUCT;
   END_VAR
BEGIN
END_DATA_BLOCK

DATA_BLOCK "DB_SystemSimu"   // DB30
// stored: Access Published, MemoryReserve 100, Namespace Global
   VAR
      TriggerSensor : Struct
         Line : Struct
            A1 : Struct
               Conveyor : Array[_.gMinA1.._.gMaxA1] of Bool;
            END_STRUCT;
            B1 : Struct
               Conveyor : Array[_.gMinB1.._.gMaxB1] of Bool;
            END_STRUCT;
            C1 : Struct
               Conveyor : Array[_.gMinC1.._.gMaxC1] of Bool;
            END_STRUCT;
            D1 : Struct
               Conveyor : Array[_.gMinD1.._.gMaxD1] of Bool;
            END_STRUCT;
         END_STRUCT;
      END_STRUCT;
      TriggerFault : Struct
         Line : Struct
            A1 : Struct
               Conveyor : Array[_.gMinA1.._.gMaxA1] of Bool;
            END_STRUCT;
            B1 : Struct
               Conveyor : Array[_.gMinB1.._.gMaxB1] of Bool;
            END_STRUCT;
            C1 : Struct
               Conveyor : Array[_.gMinC1.._.gMaxC1] of Bool;
            END_STRUCT;
            D1 : Struct
               Conveyor : Array[_.gMinD1.._.gMaxD1] of Bool;
            END_STRUCT;
         END_STRUCT;
      END_STRUCT;
      Fire : Bool;
   END_VAR
BEGIN
   // TriggerSensor.Line.A1.Conveyor[1001] : AS1.1.1
   // TriggerSensor.Line.A1.Conveyor[1002] : AS1.1.2
   // TriggerFault.Line.A1.Conveyor[1001] : AS1.1.1
   // TriggerFault.Line.A1.Conveyor[1002] : AS1.1.2
END_DATA_BLOCK

DATA_BLOCK "DB_ConveyorParameters"   // DB7
// stored: Access Published, MemoryReserve 100, Namespace Global
   VAR
      Line : Struct
         A1 : Struct
            Conveyor : Array[_.gMinA1.._.gMaxA1] of "Global.ConveyorParameters";
         END_STRUCT;
         B1 : Struct
            Conveyor : Array[_.gMinB1.._.gMaxB1] of "Global.ConveyorParameters";
         END_STRUCT;
         C1 : Struct
            Conveyor : Array[_.gMinC1.._.gMaxC1] of "Global.ConveyorParameters";
         END_STRUCT;
         D1 : Struct
            Conveyor : Array[_.gMinD1.._.gMaxD1] of "Global.ConveyorParameters";
         END_STRUCT;
      END_STRUCT;
   END_VAR
BEGIN
END_DATA_BLOCK

DATA_BLOCK "DB_Manual"   // DB22
// stored: Access Published, MemoryReserve 100, Namespace Global
   VAR
      Conveyor : Struct
         ID : Int;
         Enable : Bool;
         Run : Bool;
         in : Bool;
      END_STRUCT;
      Line : Struct
         A1 : Struct
            Conveyor { S7_SetPoint := 'True'} : Array[_.gMinA1.._.gMaxA1] of "Global.ManualInputs";
         END_STRUCT;
         B1 : Struct
            Conveyor { S7_SetPoint := 'True'} : Array[_.gMinB1.._.gMaxB1] of "Global.ManualInputs";
         END_STRUCT;
         C1 : Struct
            Conveyor { S7_SetPoint := 'True'} : Array[_.gMinC1.._.gMaxC1] of "Global.ManualInputs";
         END_STRUCT;
         D1 : Struct
            Conveyor { S7_SetPoint := 'True'} : Array[_.gMinD1.._.gMaxD1] of "Global.ManualInputs";
         END_STRUCT;
      END_STRUCT;
   END_VAR
BEGIN
END_DATA_BLOCK

DATA_BLOCK "DB_Alarm"   // DB17
// stored: Access Published, MemoryReserve 100, Namespace Global
   VAR
      "word" : Struct
         Line : Struct
            A1 : Struct
               Conveyor : Array[_.gMinA1.._.gMaxA1] of Word;
            END_STRUCT;
            B1 : Struct
               Conveyor : Array[_.gMinB1.._.gMaxB1] of Word;
            END_STRUCT;
            C1 : Struct
               Conveyor : Array[_.gMinC1.._.gMaxC1] of Word;
            END_STRUCT;
            D1 : Struct
               Conveyor : Array[_.gMinD1.._.gMaxD1] of Word;
            END_STRUCT;
         END_STRUCT;
      END_STRUCT;
      HardDiag : Struct
         ASi : Word;
         Nord : Word;
      END_STRUCT;
   END_VAR
BEGIN
END_DATA_BLOCK

DATA_BLOCK "DB_VisuColor"   // DB2
// stored: Access Published, MemoryReserve 100, Namespace Global
   VAR
      Line : Struct
         A1 : Struct
            Conveyor : Array[_.gMinA1.._.gMaxA1] of Int;
         END_STRUCT;
         B1 : Struct
            Conveyor : Array[_.gMinB1.._.gMaxB1] of Int;
         END_STRUCT;
         C1 : Struct
            Conveyor : Array[_.gMinC1.._.gMaxC1] of Int;
         END_STRUCT;
         D1 : Struct
            Conveyor : Array[_.gMinD1.._.gMaxD1] of Int;
         END_STRUCT;
      END_STRUCT;
   END_VAR
BEGIN
END_DATA_BLOCK

DATA_BLOCK "DB_ToteTracking"   // DB38
// stored: Access Published, MemoryReserve 100, Namespace Global
   VAR
      Conveyor : Array[_.gMinC1.._.gMaxC1] of "Global.TrackingData";
      Barcode : Array[_.gMinC1.._.gMaxC1] of String;
   END_VAR
BEGIN
END_DATA_BLOCK

DATA_BLOCK "DB_UDI"   // DB37
// stored: MemoryReserve 100, Namespace LineC1
   VAR
      LineC1 : Struct
         Upstream : Struct
            Conveyor : Array[_.minC1.._.maxC1] of Bool;
         END_STRUCT;
         DownstreamAccu : Struct
            Conveyor : Array[_.minC1.._.maxC1] of Bool;
         END_STRUCT;
         Interlock : Struct
            Conveyor : Array[_.minC1.._.maxC1] of Bool;
         END_STRUCT;
         Fault : Struct
            Conveyor : Array[_.minC1.._.maxC1] of Bool;
         END_STRUCT;
         Merging1 : Struct
            "Timer" : Struct
               StraightTote : TON_TIME;
               ArmTote { S7_SetPoint := 'True'} : TON_TIME;
            END_STRUCT;
            Priority : Struct
               Straight : Bool;
               Arm : Bool;
            END_STRUCT;
         END_STRUCT;
         Merging2 : Struct
            "Timer" : Struct
               StraightTote : TON_TIME;
               ArmTote { S7_SetPoint := 'True'} : TON_TIME;
            END_STRUCT;
            Priority : Struct
               Straight : Bool;
               Arm : Bool;
            END_STRUCT;
         END_STRUCT;
      END_STRUCT;
   END_VAR
BEGIN
END_DATA_BLOCK

DATA_BLOCK "DB_AsiSetpoint"   // DB32
// stored: Access Published, MemoryReserve 100, Namespace Global
   VAR
      Line : Struct
         A1 : Struct
            DirChange : Struct
               Conveyor : Array[_.gMinA1.._.gMaxA1] of Bool;
            END_STRUCT;
            Speed : Struct
               Conveyor : Array[_.gMinA1.._.gMaxA1] of Bool;
            END_STRUCT;
         END_STRUCT;
         B1 : Struct
            DirChange : Struct
               Conveyor : Array[_.gMinB1.._.gMaxB1] of Bool;
            END_STRUCT;
            Speed : Struct
               Conveyor : Array[_.gMinB1.._.gMaxB1] of Bool;
            END_STRUCT;
         END_STRUCT;
         C1 : Struct
            DirChange : Struct
               Conveyor : Array[_.gMinC1.._.gMaxC1] of Bool;
            END_STRUCT;
            Speed : Struct
               Conveyor : Array[_.gMinC1.._.gMaxC1] of Bool;
            END_STRUCT;
         END_STRUCT;
         D1 : Struct
            DirChange : Struct
               Conveyor : Array[_.gMinD1.._.gMaxD1] of Bool;
            END_STRUCT;
            Speed : Struct
               Conveyor : Array[_.gMinD1.._.gMaxD1] of Bool;
            END_STRUCT;
         END_STRUCT;
      END_STRUCT;
   END_VAR
BEGIN
   // Line.A1.DirChange.Conveyor[1001] : AS1.1.1
   // Line.A1.DirChange.Conveyor[1002] : AS1.1.2
   // Line.A1.Speed.Conveyor[1001] : AS1.1.1
   // Line.A1.Speed.Conveyor[1002] : AS1.1.2
END_DATA_BLOCK

DATA_BLOCK "DB_NordSetPoint"   // DB33
// stored: Access Published, MemoryReserve 100, Namespace Global
   VAR
      Line : Struct
         A1 : Struct   // -(0 - 16000) -> (CW: 0 - 100%) || +(0 - 16000) (CCW: 0 - 100%) || freq. has been set via NORDCON
            Conveyor : Array[_.gMinA1.._.gMaxA1] of DInt;
         END_STRUCT;
         B1 : Struct   // -(0 - 16000) -> (CW: 0 - 100%) || +(0 - 16000) (CCW: 0 - 100%) || freq. has been set via NORDCON
            Conveyor : Array[_.gMinB1.._.gMaxB1] of DInt;
         END_STRUCT;
         C1 : Struct   // -(0 - 16000) -> (CW: 0 - 100%) || +(0 - 16000) (CCW: 0 - 100%) || freq. has been set via NORDCON
            Conveyor : Array[_.gMinC1.._.gMaxC1] of DInt;
         END_STRUCT;
         D1 : Struct   // -(0 - 16000) -> (CW: 0 - 100%) || +(0 - 16000) (CCW: 0 - 100%) || freq. has been set via NORDCON
            Conveyor : Array[_.gMinD1.._.gMaxD1] of DInt;
         END_STRUCT;
      END_STRUCT;
   END_VAR
BEGIN
END_DATA_BLOCK

DATA_BLOCK "DB_S300SetPoint"   // DB21
// stored: MemoryReserve 100, Namespace Global
   VAR
      Line : Struct
         ProductionLine : Struct
            DirChange : Struct
               Conveyor : Array[_.gminProductionLine.._.gmaxProductionLine] of "Global.S300ForceMode";
            END_STRUCT;
         END_STRUCT;
      END_STRUCT;
   END_VAR
BEGIN
END_DATA_BLOCK

DATA_BLOCK "Expedtion"   // DB4
// stored: MemoryReserve 100, Namespace ProductionLine
   VAR
      ExpedtionDirection : Int;
      ExpedtionEnable : Bool;
      CurrentExpedtionDirection : String;
      StraightTableselection : Int;
      CurrentStraightTableselection : String;
      LeftTableselection : Int;
      CurrentLeftTableselection : String;
      StraightTableselectionEnable : Bool;
      LeftTableselectionEnable : Bool;
   END_VAR
BEGIN
END_DATA_BLOCK

DATA_BLOCK "DB_LogMsg"   // DB39
// stored: MemoryReserve 100, Namespace ProductionLine
   VAR
      Write_Position : Int;
      abyLogMsg_Buffer : Array[0..8191] of Byte;
      LogMsg_1 : Struct
         Para_BYTE_02 : "ProductionLine.Log_Data_Byte_Decimal";
      END_STRUCT;
      LogMsg_2 : Struct
         Para_BYTE_02 : "ProductionLine.Log_Data_Byte_Decimal";
      END_STRUCT;
      LogMsg_3 : Struct
         Para_BYTE_02 : "ProductionLine.Log_Data_Byte_Decimal";
      END_STRUCT;
      LogMsg_4 : Struct
         Para_STRING_01 : "ProductionLine.Log_Data_String20";
         Para_BYTE_02 : "ProductionLine.Log_Data_Byte_Decimal";
         Para_STRING_05 : "ProductionLine.Log_Data_String20";
      END_STRUCT;
      LogMsg_5 : Struct
         Para_STRING_01 : "ProductionLine.Log_Data_String20";
         Para_BYTE_02 : "ProductionLine.Log_Data_Byte_Decimal";
         Para_STRING_03 : "ProductionLine.Log_Data_String20";
         Para_STRING_05 : "ProductionLine.Log_Data_String20";
      END_STRUCT;
      LogMsg_6 : Struct
         Para_STRING_01 : "ProductionLine.Log_Data_String20";
         Para_BYTE_02 : "ProductionLine.Log_Data_Byte_Decimal";
      END_STRUCT;
      LogMsg_7 : Struct
         Para_STRING_01 : "ProductionLine.Log_Data_String20";
         Para_BYTE_02 : "ProductionLine.Log_Data_Byte_Decimal";
         Para_STRING_03 : "ProductionLine.Log_Data_String20";
         Para_STRING_04 : "ProductionLine.Log_Data_String20";
      END_STRUCT;
      LogMsg_8 : Struct
         Para_STRING_01 : "ProductionLine.Log_Data_String20";
         Para_BYTE_02 : "ProductionLine.Log_Data_Byte_Decimal";
      END_STRUCT;
      LogMsg_9 : Struct
         Para_STRING_01 : "ProductionLine.Log_Data_String20";
         Para_BYTE_02 : "ProductionLine.Log_Data_Byte_Decimal";
         Para_STRING_03 : "ProductionLine.Log_Data_String20";
         Para_STRING_04 : "ProductionLine.Log_Data_String20";
         Para_STRING_05 : "ProductionLine.Log_Data_String20";
      END_STRUCT;
      LogMsg_10 : Struct
         Para_STRING_01 : "ProductionLine.Log_Data_String20";
         Para_BYTE_02 : "ProductionLine.Log_Data_Byte_Decimal";
         Para_STRING_03 : "ProductionLine.Log_Data_String20";
         Para_STRING_04 : "ProductionLine.Log_Data_String20";
         Para_CHAR_05 : "ProductionLine.Log_Data_Char";
      END_STRUCT;
   END_VAR
BEGIN
END_DATA_BLOCK

DATA_BLOCK "OPC_Data"   // DB41
// stored: MemoryReserve 0, Namespace ProductionLine
   VAR
      Watchdog : Struct
         Keep_Alive_PLC : Int;   // //Periodic counter, incremented every 10 seconds. If one side does not increment the counter within 30 seconds, it will be considered offline by the other side.
         Keep_Alive_WMS : Int;   // //Periodic counter, incremented every 10 seconds. If one side does not increment the counter within 30 seconds, it will be considered offline by the other side.
      END_STRUCT;
      DP1 : Struct
         DestRequest : Struct
            Source : "ProductionLine.OPC_DsetRequest";
            Ack { S7_SetPoint := 'True'} : "ProductionLine.OPC_DestRequest_Ack";
         END_STRUCT;
      END_STRUCT;
      DP2 : Struct
         DestRequest : Struct
            Source : "ProductionLine.OPC_DsetRequest";
            Ack { S7_SetPoint := 'True'} : "ProductionLine.OPC_DestRequest_Ack";
         END_STRUCT;
      END_STRUCT;
      DP3 : Struct
         DestRequest : Struct
            Source : "ProductionLine.OPC_DsetRequest";
            Ack { S7_SetPoint := 'True'} : "ProductionLine.OPC_DestRequest_Ack";
         END_STRUCT;
      END_STRUCT;
      DP4 : Struct
         DestRequest : Struct
            Source : "ProductionLine.OPC_DsetRequest";
            Ack { S7_SetPoint := 'True'} : "ProductionLine.OPC_DestRequest_Ack";
         END_STRUCT;
      END_STRUCT;
      IP11 : Struct
         DestInfo : Struct
            Source : "ProductionLine.OPC_DestInfo";
            Ack { S7_SetPoint := 'True'} : "ProductionLine.OPC_DestInfo_Ack";
         END_STRUCT;
      END_STRUCT;
      IP12 : Struct
         DestInfo : Struct
            Source : "ProductionLine.OPC_DestInfo";
            Ack { S7_SetPoint := 'True'} : "ProductionLine.OPC_DestInfo_Ack";
         END_STRUCT;
      END_STRUCT;
      IP21 : Struct
         DestInfo : Struct
            Source : "ProductionLine.OPC_DestInfo";
            Ack { S7_SetPoint := 'True'} : "ProductionLine.OPC_DestInfo_Ack";
         END_STRUCT;
      END_STRUCT;
      IP22 : Struct
         DestInfo : Struct
            Source : "ProductionLine.OPC_DestInfo";
            Ack { S7_SetPoint := 'True'} : "ProductionLine.OPC_DestInfo_Ack";
         END_STRUCT;
      END_STRUCT;
      IP23 : Struct
         DestInfo : Struct
            Source : "ProductionLine.OPC_DestInfo";
            Ack { S7_SetPoint := 'True'} : "ProductionLine.OPC_DestInfo_Ack";
         END_STRUCT;
      END_STRUCT;
      IP31 : Struct
         DestInfo : Struct
            Source : "ProductionLine.OPC_DestInfo";
            Ack { S7_SetPoint := 'True'} : "ProductionLine.OPC_DestInfo_Ack";
         END_STRUCT;
      END_STRUCT;
      IP32 : Struct
         DestInfo : Struct
            Source : "ProductionLine.OPC_DestInfo";
            Ack { S7_SetPoint := 'True'} : "ProductionLine.OPC_DestInfo_Ack";
         END_STRUCT;
      END_STRUCT;
      IP41 : Struct
         DestInfo : Struct
            Source : "ProductionLine.OPC_DestInfo";
            Ack { S7_SetPoint := 'True'} : "ProductionLine.OPC_DestInfo_Ack";
         END_STRUCT;
      END_STRUCT;
      IP42 : Struct
         DestInfo : Struct
            Source : "ProductionLine.OPC_DestInfo";
            Ack { S7_SetPoint := 'True'} : "ProductionLine.OPC_DestInfo_Ack";
         END_STRUCT;
      END_STRUCT;
      Status : "ProductionLine.OPC_SegmentStatus";
   END_VAR
BEGIN
   DP1.DestRequest.Source.DecisionPoint := 'DP1';
   DP2.DestRequest.Source.DecisionPoint := 'DP2';
   DP3.DestRequest.Source.DecisionPoint := 'DP3';
   DP4.DestRequest.Source.DecisionPoint := 'DP4';
   IP11.DestInfo.Source.DecisionPoint := 'DP1';
   IP12.DestInfo.Source.DecisionPoint := 'DP1';
   IP21.DestInfo.Source.DecisionPoint := 'DP2';
   IP22.DestInfo.Source.DecisionPoint := 'DP2';
   IP23.DestInfo.Source.DecisionPoint := 'DP2';
   IP31.DestInfo.Source.DecisionPoint := 'DP3';
   IP32.DestInfo.Source.DecisionPoint := 'DP3';
   IP41.DestInfo.Source.DecisionPoint := 'DP4';
   IP42.DestInfo.Source.DecisionPoint := 'DP4';
END_DATA_BLOCK

ORGANIZATION_BLOCK "Main"   // OB1, LAD, ProgramCycle
TITLE = "Main Program Sweep (Cycle)"
{ S7_Optimized_Access := 'TRUE' }
// stored: SetENOAutomatically false
   VAR_INPUT
      Initial_Call : Bool;   // Initial call of this OB
      Remanence : Bool;   // =True, if remanent data are available
   END_VAR
BEGIN

REGION Network 1
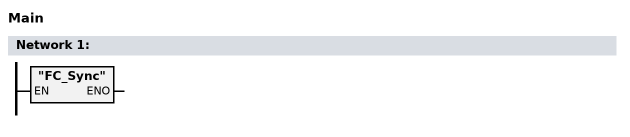
   RUNG wire#powerrail
      "FC_Sync"()
   END_RUNG
   // the same network as SCL:
   "FC_Sync"();
END_REGION
END_ORGANIZATION_BLOCK

FUNCTION "FC_Sync" : Void
{ S7_Optimized_Access := 'TRUE' }
VERSION : 0.1

BEGIN
	
	
	
	REGION system memory bits
	    
	    "DB_Sync".memoryBit.System_Byte := "System_Byte";
	    "DB_Sync".memoryBit.FirstScan := "FirstScan";
	    "DB_Sync".memoryBit.DiagStatusUpdate := "DiagStatusUpdate";
	    "DB_Sync".memoryBit.AlwaysTRUE := "AlwaysTRUE";
	    "DB_Sync".memoryBit.AlwaysFALSE := "AlwaysFALSE";
	    
	END_REGION
	
	REGION clock memory bits
	    
	    "DB_Sync".ClockBit.Clock_Byte := "Clock_Byte";
	    "DB_Sync".ClockBit."Clock_10Hz" := "Clock_10Hz";
	    "DB_Sync".ClockBit."Clock_5Hz" := "Clock_5Hz";
	    "DB_Sync".ClockBit."Clock_2.5Hz" := "Clock_2.5Hz";
	    "DB_Sync".ClockBit."Clock_2Hz" := "Clock_2Hz";
	    "DB_Sync".ClockBit."Clock_1.25Hz" := "Clock_1.25Hz";
	    "DB_Sync".ClockBit."Clock_1Hz" := "Clock_1Hz";
	    "DB_Sync".ClockBit."Clock_0.625Hz" := "Clock_0.625Hz";
	    "DB_Sync".ClockBit."Clock_0.5Hz" := "Clock_0.5Hz";
	    
	END_REGION
	
	REGION System tsrat/stop
	    // Statement section REGION
	    "DB_Sync".startbit := "startBit";
	    "DB_Sync".stopbit := "stopBit";
	    "DB_Sync".resetbit := "ResetBit";
	    
	END_REGION
	
	
	
	
	
	
	
	
	
	
	
	
	
	
	
	
END_FUNCTION

FUNCTION_BLOCK "FSFB_Main_Safety_RTG1"   // FB1, F_FBD
   VAR
      ESTOP : ESTOP1;
   END_VAR
BEGIN

REGION Network 1
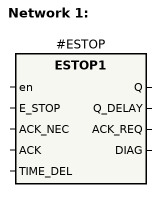
   #ESTOP();   // ESTOP1
END_REGION
END_FUNCTION_BLOCK

FUNCTION_BLOCK "FB_AutoReset"   // FB21, LAD
// stored: Access Published, MemoryReserve 100, Namespace Global, SetENOAutomatically false
   VAR_INPUT
      AckIN : Bool;
   END_VAR
   VAR_OUTPUT
      Ack : Bool;
   END_VAR
   VAR
      MemoryBit : Array[1..2] of Bool;
      "Timer" { S7_SetPoint := 'True'} : TOF_TIME;
   END_VAR
   VAR_TEMP   // added for the SCL form of the ladder/FBD networks
      _w1 : Bool;
      _w2 : Bool;
   END_VAR
BEGIN

REGION Network 1
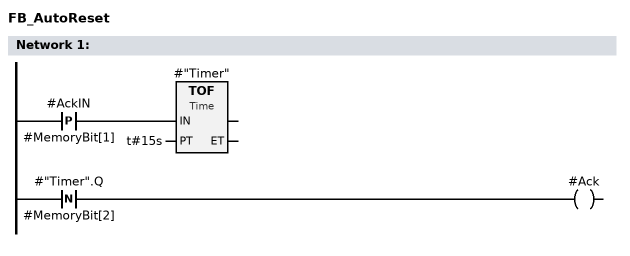
   RUNG wire#powerrail
      P_Contact(operand := #AckIN, bit := #MemoryBit[1])
      { S7_Templates := "time_type := Time" } #"Timer".TOF(pt := t#15s, et =>)
   END_RUNG
   RUNG wire#powerrail
      N_Contact(operand := #"Timer".Q, bit := #MemoryBit[2])
      Coil( #Ack )
   END_RUNG
   // the same network as SCL:
   #_w1 := #AckIN AND NOT #MemoryBit[1];   // rising edge of #AckIN
   #MemoryBit[1] := #AckIN;
   #"Timer"(IN := #_w1, PT := t#15s);   // TOF
   #_w2 := NOT #"Timer".Q AND #MemoryBit[2];   // falling edge of #"Timer".Q
   #MemoryBit[2] := #"Timer".Q;
   #Ack := #_w2;
END_REGION
END_FUNCTION_BLOCK

FUNCTION "FC_ManualSorter" : Void   // FC18, LAD
// stored: Access Published, Namespace Global, SetENOAutomatically false
   VAR_INPUT
      RunWheels : Bool;
      "GoRight/left" : Bool;
      GoStraight : Bool;
      "positionRight/Left" : Bool;
      positionStraight : Bool;
   END_VAR
   VAR_OUTPUT
      CmdRunWheels : Bool;
      "CmdRight/Left" : Bool;
      CmdStraight : Bool;
   END_VAR
BEGIN

REGION Network 1: status manual
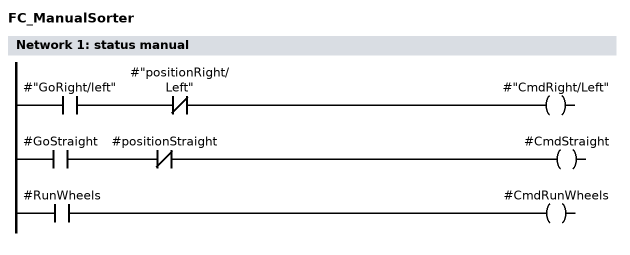
   RUNG wire#powerrail
      Contact( #"GoRight/left" )
      I_Contact( #"positionRight/Left" )
      Coil( #"CmdRight/Left" )
   END_RUNG
   RUNG wire#powerrail
      Contact( #GoStraight )
      I_Contact( #positionStraight )
      Coil( #CmdStraight )
   END_RUNG
   RUNG wire#powerrail
      Contact( #RunWheels )
      Coil( #CmdRunWheels )
   END_RUNG
   // the same network as SCL:
   #"CmdRight/Left" := #"GoRight/left" AND NOT #"positionRight/Left";
   #CmdStraight := #GoStraight AND NOT #positionStraight;
   #CmdRunWheels := #RunWheels;
END_REGION
END_FUNCTION

FUNCTION "FC_ManualStopper" : Void   // FC13, LAD
// stored: Access Published, Namespace Global, SetENOAutomatically false
   VAR_INPUT
      GoUp : Bool;
      GoDown : Bool;
      positionUp : Bool;
      positionDown : Bool;
   END_VAR
   VAR_OUTPUT
      CmdUP : Bool;
      cmdDOWN : Bool;
   END_VAR
BEGIN

REGION Network 1: status manual
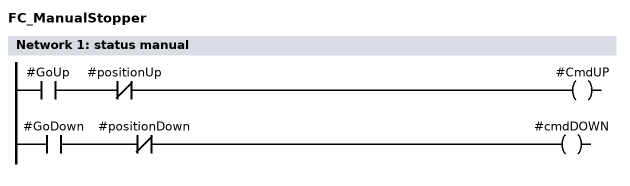
   RUNG wire#powerrail
      Contact( #GoUp )
      I_Contact( #positionUp )
      Coil( #CmdUP )
   END_RUNG
   RUNG wire#powerrail
      Contact( #GoDown )
      I_Contact( #positionDown )
      Coil( #cmdDOWN )
   END_RUNG
   // the same network as SCL:
   #CmdUP := #GoUp AND NOT #positionUp;
   #cmdDOWN := #GoDown AND NOT #positionDown;
END_REGION
END_FUNCTION

FUNCTION_BLOCK "FB_MABS_PNIO"   // FB6, LAD
// stored: Access Published, MemoryReserve 100, Namespace Global, SetENOAutomatically false
   VAR_IN_OUT
      IBP_in : "IB_P01/02/03_in_64bytes_struct";
      IBP_out : "IB_P01/02/03_out_64bytes_struct";
      MABS : "Global.MABS";
   END_VAR
   VAR
      Initializing : Bool;
      Waiting_sw_req : Bool;
      Switching_left : Bool;
      "Switching_left to straight" : Bool;
      "Switching_right to straight" : Bool;
      Switching_right : Bool;
      Switching_done : Bool;
      Tof_life_bit { S7_SetPoint := 'True'} : TON_TIME;
      MABS_sw_timout { S7_SetPoint := 'True'} : TON_TIME;
      "position status_right" : Bool;
      "position status_left" : Bool;
      "position status_straight" : Bool;
      Edge0 : Bool;
      Edge1 : Bool;
      Edge2 : Bool;
      Edge3 : Bool;
      Edge4 : Bool;
      Edge5 : Bool;
      Edge6 : Bool;
      Ton_err_motor_A { S7_SetPoint := 'True'} : TON_TIME;
      Ton_err_motor_B { S7_SetPoint := 'True'} : TON_TIME;
      Ton_err_motor_Com { S7_SetPoint := 'True'} : TON_TIME;
   END_VAR
   VAR_TEMP
      Temp_err_com : Bool;
   END_VAR
   VAR_TEMP   // added for the SCL form of the ladder/FBD networks
      _w1 : Bool;
      _w2 : Bool;
   END_VAR
BEGIN

REGION Network 1: Error motor A & B
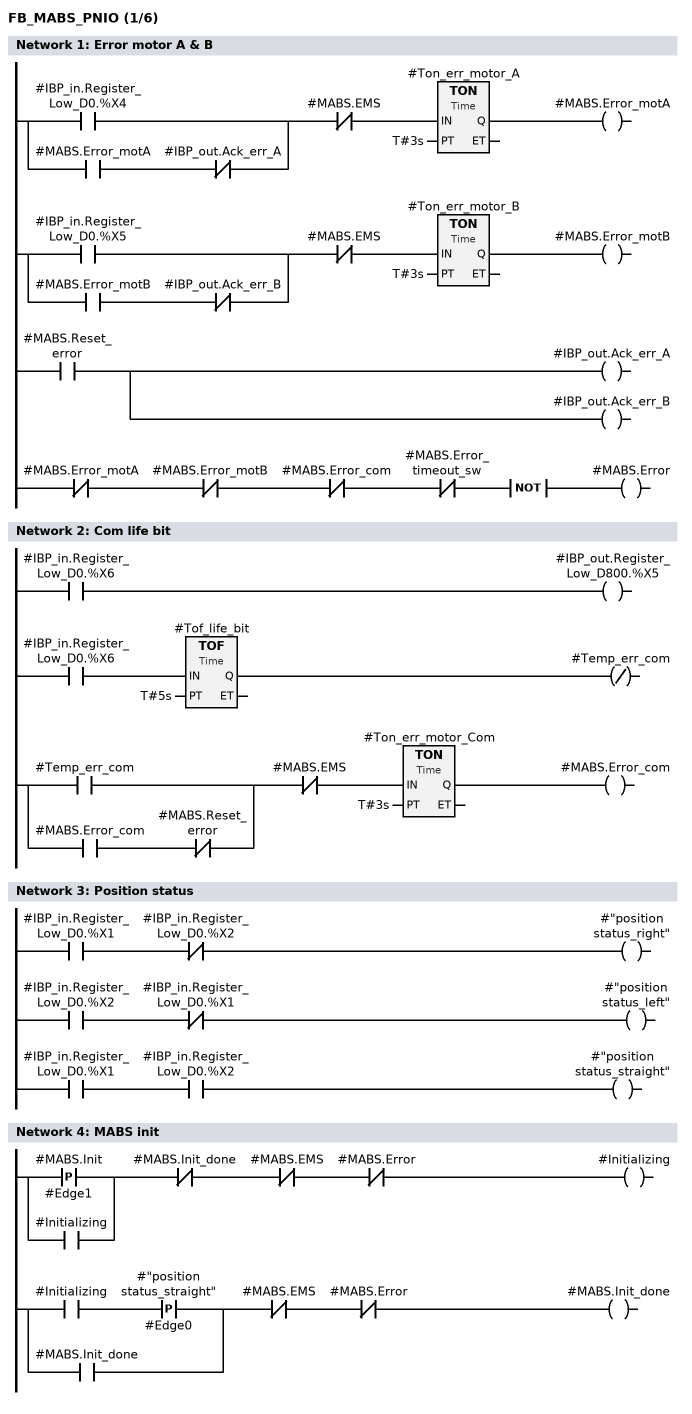
   RUNG wire#powerrail
      Contact( #IBP_in.Register_Low_D0.%X4 )
      wire#w1
      I_Contact( #MABS.EMS )
      { S7_Templates := "time_type := Time" } #Ton_err_motor_A.TON(pt := T#3s, et =>)
      Coil( #MABS.Error_motA )
   END_RUNG
   RUNG wire#powerrail
      Contact( #MABS.Error_motA )
      I_Contact( #IBP_out.Ack_err_A )
   END_RUNG wire#w1
   RUNG wire#powerrail
      Contact( #IBP_in.Register_Low_D0.%X5 )
      wire#w2
      I_Contact( #MABS.EMS )
      { S7_Templates := "time_type := Time" } #Ton_err_motor_B.TON(pt := T#3s, et =>)
      Coil( #MABS.Error_motB )
   END_RUNG
   RUNG wire#powerrail
      Contact( #MABS.Error_motB )
      I_Contact( #IBP_out.Ack_err_B )
   END_RUNG wire#w2
   RUNG wire#powerrail
      Contact( #MABS.Reset_error )
      wire#w3
      Coil( #IBP_out.Ack_err_A )
   END_RUNG
   RUNG wire#w3
      Coil( #IBP_out.Ack_err_B )
   END_RUNG
   RUNG wire#powerrail
      I_Contact( #MABS.Error_motA )
      I_Contact( #MABS.Error_motB )
      I_Contact( #MABS.Error_com )
      I_Contact( #MABS.Error_timeout_sw )
      Not()
      Coil( #MABS.Error )
   END_RUNG
   // the same network as SCL:
   #Ton_err_motor_A(IN := (#IBP_in.Register_Low_D0.%X4 OR (#MABS.Error_motA AND NOT #IBP_out.Ack_err_A)) AND NOT #MABS.EMS,   // TON
                    PT := T#3s);
   #MABS.Error_motA := #Ton_err_motor_A.Q;
   #Ton_err_motor_B(IN := (#IBP_in.Register_Low_D0.%X5 OR (#MABS.Error_motB AND NOT #IBP_out.Ack_err_B)) AND NOT #MABS.EMS,   // TON
                    PT := T#3s);
   #MABS.Error_motB := #Ton_err_motor_B.Q;
   #IBP_out.Ack_err_A := #MABS.Reset_error;
   #IBP_out.Ack_err_B := #MABS.Reset_error;
   #MABS.Error := NOT (NOT #MABS.Error_motA AND NOT #MABS.Error_motB AND NOT #MABS.Error_com AND NOT #MABS.Error_timeout_sw);
END_REGION

REGION Network 2: Com life bit
   RUNG wire#powerrail
      Contact( #IBP_in.Register_Low_D0.%X6 )
      Coil( #IBP_out.Register_Low_D800.%X5 )
   END_RUNG
   RUNG wire#powerrail
      Contact( #IBP_in.Register_Low_D0.%X6 )
      { S7_Templates := "time_type := Time" } #Tof_life_bit.TOF(pt := T#5s, et =>)
      I_Coil( #Temp_err_com )
   END_RUNG
   RUNG wire#powerrail
      Contact( #Temp_err_com )
      wire#w1
      I_Contact( #MABS.EMS )
      { S7_Templates := "time_type := Time" } #Ton_err_motor_Com.TON(pt := T#3s, et =>)
      Coil( #MABS.Error_com )
   END_RUNG
   RUNG wire#powerrail
      Contact( #MABS.Error_com )
      I_Contact( #MABS.Reset_error )
   END_RUNG wire#w1
   // the same network as SCL:
   #IBP_out.Register_Low_D800.%X5 := #IBP_in.Register_Low_D0.%X6;
   #Tof_life_bit(IN := #IBP_in.Register_Low_D0.%X6, PT := T#5s);   // TOF
   #Temp_err_com := NOT #Tof_life_bit.Q;
   #Ton_err_motor_Com(IN := (#Temp_err_com OR (#MABS.Error_com AND NOT #MABS.Reset_error)) AND NOT #MABS.EMS,   // TON
                      PT := T#3s);
   #MABS.Error_com := #Ton_err_motor_Com.Q;
END_REGION

REGION Network 3: Position status
   RUNG wire#powerrail
      Contact( #IBP_in.Register_Low_D0.%X1 )
      I_Contact( #IBP_in.Register_Low_D0.%X2 )
      Coil( #"position status_right" )
   END_RUNG
   RUNG wire#powerrail
      Contact( #IBP_in.Register_Low_D0.%X2 )
      I_Contact( #IBP_in.Register_Low_D0.%X1 )
      Coil( #"position status_left" )
   END_RUNG
   RUNG wire#powerrail
      Contact( #IBP_in.Register_Low_D0.%X1 )
      Contact( #IBP_in.Register_Low_D0.%X2 )
      Coil( #"position status_straight" )
   END_RUNG
   // the same network as SCL:
   #"position status_right" := #IBP_in.Register_Low_D0.%X1 AND NOT #IBP_in.Register_Low_D0.%X2;
   #"position status_left" := #IBP_in.Register_Low_D0.%X2 AND NOT #IBP_in.Register_Low_D0.%X1;
   #"position status_straight" := #IBP_in.Register_Low_D0.%X1 AND #IBP_in.Register_Low_D0.%X2;
END_REGION

REGION Network 4: MABS init
   RUNG wire#powerrail
      P_Contact(operand := #MABS.Init, bit := #Edge1)
      wire#w1
      I_Contact( #MABS.Init_done )
      I_Contact( #MABS.EMS )
      I_Contact( #MABS.Error )
      Coil( #Initializing )
   END_RUNG
   RUNG wire#powerrail
      Contact( #Initializing )
   END_RUNG wire#w1
   RUNG wire#powerrail
      Contact( #Initializing )
      P_Contact(operand := #"position status_straight", bit := #Edge0)
      wire#w2
      I_Contact( #MABS.EMS )
      I_Contact( #MABS.Error )
      Coil( #MABS.Init_done )
   END_RUNG
   RUNG wire#powerrail
      Contact( #MABS.Init_done )
   END_RUNG wire#w2
   // the same network as SCL:
   #_w1 := #MABS.Init AND NOT #Edge1;   // rising edge of #MABS.Init
   #Edge1 := #MABS.Init;
   #Initializing := (#_w1 OR #Initializing) AND NOT #MABS.Init_done AND NOT #MABS.EMS AND NOT #MABS.Error;
   #_w2 := #Initializing AND #"position status_straight" AND NOT #Edge0;   // rising edge of #"position status_straight"
   #Edge0 := #"position status_straight";
   #MABS.Init_done := (#_w2 OR #MABS.Init_done) AND NOT #MABS.EMS AND NOT #MABS.Error;
END_REGION

REGION Network 5: MABS ready
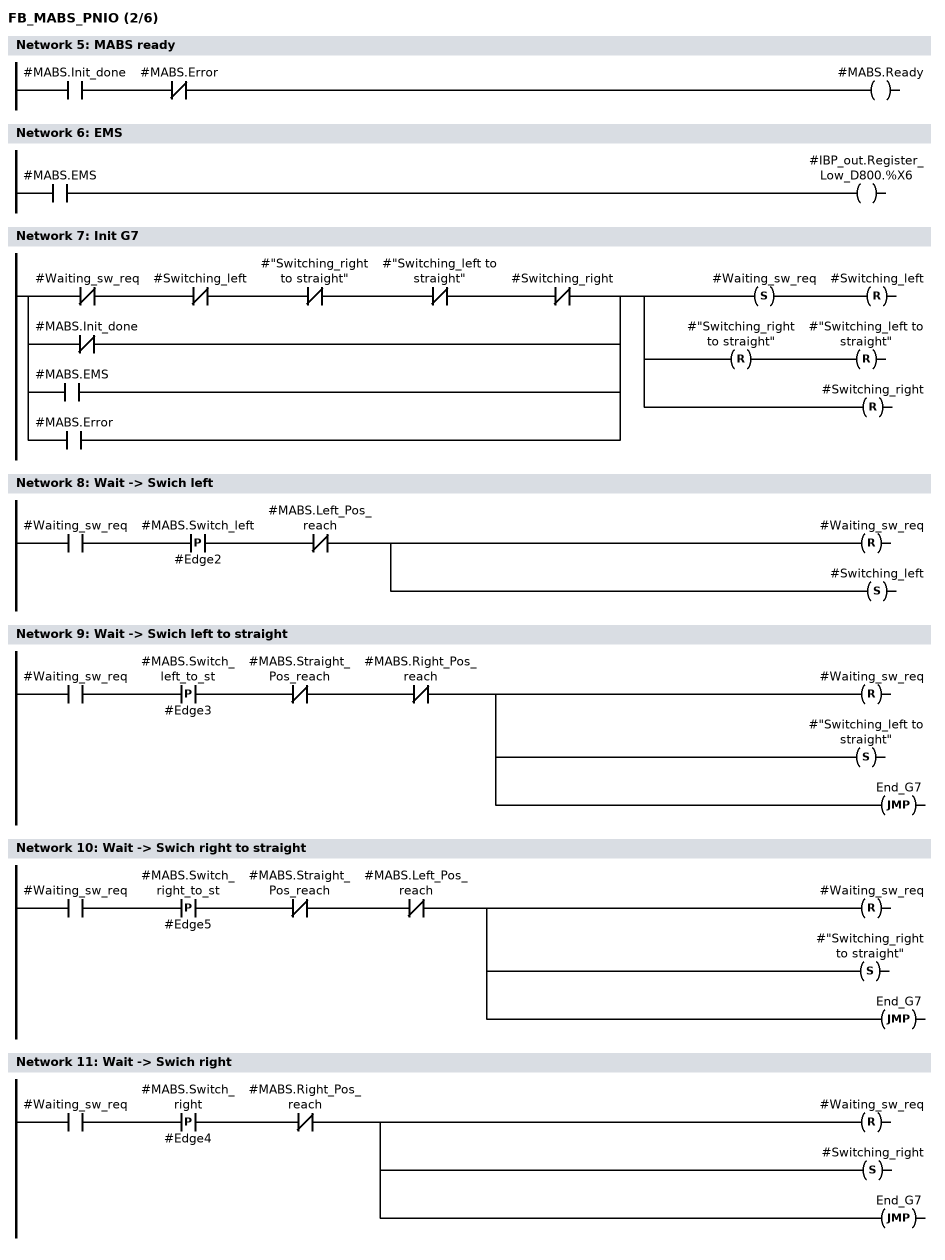
   RUNG wire#powerrail
      Contact( #MABS.Init_done )
      I_Contact( #MABS.Error )
      Coil( #MABS.Ready )
   END_RUNG
   // the same network as SCL:
   #MABS.Ready := #MABS.Init_done AND NOT #MABS.Error;
END_REGION

REGION Network 6: EMS
   RUNG wire#powerrail
      Contact( #MABS.EMS )
      Coil( #IBP_out.Register_Low_D800.%X6 )
   END_RUNG
   // the same network as SCL:
   #IBP_out.Register_Low_D800.%X6 := #MABS.EMS;
END_REGION

REGION Network 7: Init G7
   RUNG wire#powerrail
      I_Contact( #Waiting_sw_req )
      I_Contact( #Switching_left )
      I_Contact( #"Switching_right to straight" )
      I_Contact( #"Switching_left to straight" )
      I_Contact( #Switching_right )
      wire#w1
      S_Coil( #Waiting_sw_req )
      R_Coil( #Switching_left )
   END_RUNG
   RUNG wire#powerrail
      I_Contact( #MABS.Init_done )
   END_RUNG wire#w1
   RUNG wire#powerrail
      Contact( #MABS.EMS )
   END_RUNG wire#w1
   RUNG wire#powerrail
      Contact( #MABS.Error )
   END_RUNG wire#w1
   RUNG wire#w1
      R_Coil( #"Switching_right to straight" )
      R_Coil( #"Switching_left to straight" )
   END_RUNG
   RUNG wire#w1
      R_Coil( #Switching_right )
   END_RUNG
   // the same network as SCL:
   #_w1 := (NOT #Waiting_sw_req AND NOT #Switching_left AND NOT #"Switching_right to straight" AND NOT #"Switching_left to straight" AND NOT #Switching_right) OR NOT #MABS.Init_done OR #MABS.EMS OR #MABS.Error;
   IF #_w1 THEN
       #Waiting_sw_req := TRUE;
       #Switching_left := FALSE;
       #"Switching_right to straight" := FALSE;
       #"Switching_left to straight" := FALSE;
       #Switching_right := FALSE;
   END_IF;
END_REGION

REGION Network 8: Wait -> Swich left
   RUNG wire#powerrail
      Contact( #Waiting_sw_req )
      P_Contact(operand := #MABS.Switch_left, bit := #Edge2)
      I_Contact( #MABS.Left_Pos_reach )
      wire#w1
      R_Coil( #Waiting_sw_req )
   END_RUNG
   RUNG wire#w1
      S_Coil( #Switching_left )
   END_RUNG
   // the same network as SCL:
   #_w1 := #Waiting_sw_req AND #MABS.Switch_left AND NOT #Edge2;   // rising edge of #MABS.Switch_left
   #Edge2 := #MABS.Switch_left;
   IF #_w1 AND NOT #MABS.Left_Pos_reach THEN
       #Waiting_sw_req := FALSE;
       #Switching_left := TRUE;
   END_IF;
END_REGION

REGION Network 9: Wait -> Swich left to straight
   RUNG wire#powerrail
      Contact( #Waiting_sw_req )
      P_Contact(operand := #MABS.Switch_left_to_st, bit := #Edge3)
      I_Contact( #MABS.Straight_Pos_reach )
      I_Contact( #MABS.Right_Pos_reach )
      wire#w1
      R_Coil( #Waiting_sw_req )
   END_RUNG
   RUNG wire#w1
      S_Coil( #"Switching_left to straight" )
   END_RUNG
   RUNG wire#w1
      JumpCoil( End_G7 )
   END_RUNG
   // the same network as SCL:
   #_w1 := #Waiting_sw_req AND #MABS.Switch_left_to_st AND NOT #Edge3;   // rising edge of #MABS.Switch_left_to_st
   #Edge3 := #MABS.Switch_left_to_st;
   #_w2 := #_w1 AND NOT #MABS.Straight_Pos_reach AND NOT #MABS.Right_Pos_reach;
   IF #_w2 THEN
       #Waiting_sw_req := FALSE;
       #"Switching_left to straight" := TRUE;
       GOTO End_G7;
   END_IF;
END_REGION

REGION Network 10: Wait -> Swich right to straight
   RUNG wire#powerrail
      Contact( #Waiting_sw_req )
      P_Contact(operand := #MABS.Switch_right_to_st, bit := #Edge5)
      I_Contact( #MABS.Straight_Pos_reach )
      I_Contact( #MABS.Left_Pos_reach )
      wire#w1
      R_Coil( #Waiting_sw_req )
   END_RUNG
   RUNG wire#w1
      S_Coil( #"Switching_right to straight" )
   END_RUNG
   RUNG wire#w1
      JumpCoil( End_G7 )
   END_RUNG
   // the same network as SCL:
   #_w1 := #Waiting_sw_req AND #MABS.Switch_right_to_st AND NOT #Edge5;   // rising edge of #MABS.Switch_right_to_st
   #Edge5 := #MABS.Switch_right_to_st;
   #_w2 := #_w1 AND NOT #MABS.Straight_Pos_reach AND NOT #MABS.Left_Pos_reach;
   IF #_w2 THEN
       #Waiting_sw_req := FALSE;
       #"Switching_right to straight" := TRUE;
       GOTO End_G7;
   END_IF;
END_REGION

REGION Network 11: Wait -> Swich right
   RUNG wire#powerrail
      Contact( #Waiting_sw_req )
      P_Contact(operand := #MABS.Switch_right, bit := #Edge4)
      I_Contact( #MABS.Right_Pos_reach )
      wire#w1
      R_Coil( #Waiting_sw_req )
   END_RUNG
   RUNG wire#w1
      S_Coil( #Switching_right )
   END_RUNG
   RUNG wire#w1
      JumpCoil( End_G7 )
   END_RUNG
   // the same network as SCL:
   #_w1 := #Waiting_sw_req AND #MABS.Switch_right AND NOT #Edge4;   // rising edge of #MABS.Switch_right
   #Edge4 := #MABS.Switch_right;
   #_w2 := #_w1 AND NOT #MABS.Right_Pos_reach;
   IF #_w2 THEN
       #Waiting_sw_req := FALSE;
       #Switching_right := TRUE;
       GOTO End_G7;
   END_IF;
END_REGION

REGION Network 12: Swich right -> Wait
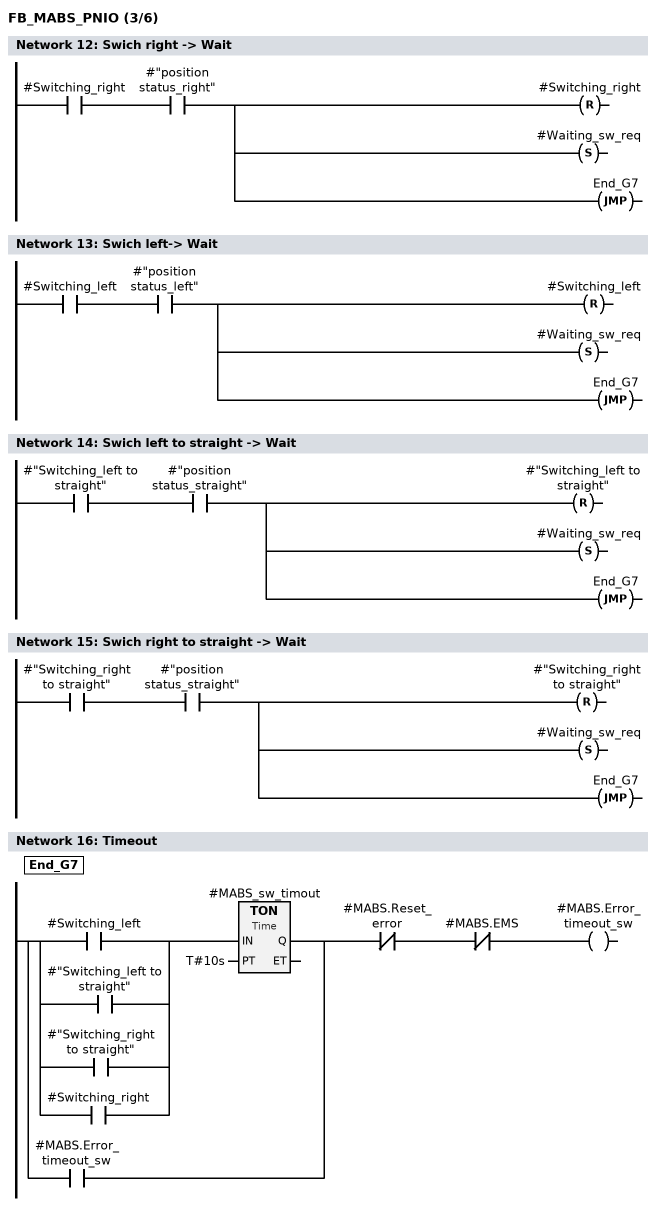
   RUNG wire#powerrail
      Contact( #Switching_right )
      Contact( #"position status_right" )
      wire#w1
      R_Coil( #Switching_right )
   END_RUNG
   RUNG wire#w1
      S_Coil( #Waiting_sw_req )
   END_RUNG
   RUNG wire#w1
      JumpCoil( End_G7 )
   END_RUNG
   // the same network as SCL:
   #_w1 := #Switching_right AND #"position status_right";
   IF #_w1 THEN
       #Switching_right := FALSE;
       #Waiting_sw_req := TRUE;
       GOTO End_G7;
   END_IF;
END_REGION

REGION Network 13: Swich left-> Wait
   RUNG wire#powerrail
      Contact( #Switching_left )
      Contact( #"position status_left" )
      wire#w1
      R_Coil( #Switching_left )
   END_RUNG
   RUNG wire#w1
      S_Coil( #Waiting_sw_req )
   END_RUNG
   RUNG wire#w1
      JumpCoil( End_G7 )
   END_RUNG
   // the same network as SCL:
   #_w1 := #Switching_left AND #"position status_left";
   IF #_w1 THEN
       #Switching_left := FALSE;
       #Waiting_sw_req := TRUE;
       GOTO End_G7;
   END_IF;
END_REGION

REGION Network 14: Swich left to straight -> Wait
   RUNG wire#powerrail
      Contact( #"Switching_left to straight" )
      Contact( #"position status_straight" )
      wire#w1
      R_Coil( #"Switching_left to straight" )
   END_RUNG
   RUNG wire#w1
      S_Coil( #Waiting_sw_req )
   END_RUNG
   RUNG wire#w1
      JumpCoil( End_G7 )
   END_RUNG
   // the same network as SCL:
   #_w1 := #"Switching_left to straight" AND #"position status_straight";
   IF #_w1 THEN
       #"Switching_left to straight" := FALSE;
       #Waiting_sw_req := TRUE;
       GOTO End_G7;
   END_IF;
END_REGION

REGION Network 15: Swich right to straight -> Wait
   RUNG wire#powerrail
      Contact( #"Switching_right to straight" )
      Contact( #"position status_straight" )
      wire#w1
      R_Coil( #"Switching_right to straight" )
   END_RUNG
   RUNG wire#w1
      S_Coil( #Waiting_sw_req )
   END_RUNG
   RUNG wire#w1
      JumpCoil( End_G7 )
   END_RUNG
   // the same network as SCL:
   #_w1 := #"Switching_right to straight" AND #"position status_straight";
   IF #_w1 THEN
       #"Switching_right to straight" := FALSE;
       #Waiting_sw_req := TRUE;
       GOTO End_G7;
   END_IF;
END_REGION

